IF SUPER^.Step(746, TRUE, 'Step number 746') THEN
    SUPER^.StepCompleteWhen((_runOneStep OR _runAllSteps) AND _finishStep);

    IF _runOneStep THEN
        _runOneStep := FALSE;
        RETURN;
    END_IF
END_IF

IF SUPER^.Step(747, TRUE, 'Step number 747') THEN
    SUPER^.StepCompleteWhen((_runOneStep OR _runAllSteps) AND _finishStep);

    IF _runOneStep THEN
        _runOneStep := FALSE;
        RETURN;
    END_IF
END_IF

IF SUPER^.Step(748, TRUE, 'Step number 748') THEN
    SUPER^.StepCompleteWhen((_runOneStep OR _runAllSteps) AND _finishStep);

    IF _runOneStep THEN
        _runOneStep := FALSE;
        RETURN;
    END_IF
END_IF

IF SUPER^.Step(749, TRUE, 'Step number 749') THEN
    SUPER^.StepCompleteWhen((_runOneStep OR _runAllSteps) AND _finishStep);

    IF _runOneStep THEN
        _runOneStep := FALSE;
        RETURN;
    END_IF
END_IF

IF SUPER^.Step(750, TRUE, 'Step number 750') THEN
    SUPER^.StepCompleteWhen((_runOneStep OR _runAllSteps) AND _finishStep);

    IF _runOneStep THEN
        _runOneStep := FALSE;
        RETURN;
    END_IF
END_IF

IF SUPER^.Step(751, TRUE, 'Step number 751') THEN
    SUPER^.StepCompleteWhen((_runOneStep OR _runAllSteps) AND _finishStep);

    IF _runOneStep THEN
        _runOneStep := FALSE;
        RETURN;
    END_IF
END_IF

IF SUPER^.Step(752, TRUE, 'Step number 752') THEN
    SUPER^.StepCompleteWhen((_runOneStep OR _runAllSteps) AND _finishStep);

    IF _runOneStep THEN
        _runOneStep := FALSE;
        RETURN;
    END_IF
END_IF

IF SUPER^.Step(753, TRUE, 'Step number 753') THEN
    SUPER^.StepCompleteWhen((_runOneStep OR _runAllSteps) AND _finishStep);

    IF _runOneStep THEN
        _runOneStep := FALSE;
        RETURN;
    END_IF
END_IF

IF SUPER^.Step(754, TRUE, 'Step number 754') THEN
    SUPER^.StepCompleteWhen((_runOneStep OR _runAllSteps) AND _finishStep);

    IF _runOneStep THEN
        _runOneStep := FALSE;
        RETURN;
    END_IF
END_IF

IF SUPER^.Step(755, TRUE, 'Step number 755') THEN
    SUPER^.StepCompleteWhen((_runOneStep OR _runAllSteps) AND _finishStep);

    IF _runOneStep THEN
        _runOneStep := FALSE;
        RETURN;
    END_IF
END_IF

IF SUPER^.Step(756, TRUE, 'Step number 756') THEN
    SUPER^.StepCompleteWhen((_runOneStep OR _runAllSteps) AND _finishStep);

    IF _runOneStep THEN
        _runOneStep := FALSE;
        RETURN;
    END_IF
END_IF

IF SUPER^.Step(757, TRUE, 'Step number 757') THEN
    SUPER^.StepCompleteWhen((_runOneStep OR _runAllSteps) AND _finishStep);

    IF _runOneStep THEN
        _runOneStep := FALSE;
        RETURN;
    END_IF
END_IF

IF SUPER^.Step(758, TRUE, 'Step number 758') THEN
    SUPER^.StepCompleteWhen((_runOneStep OR _runAllSteps) AND _finishStep);

    IF _runOneStep THEN
        _runOneStep := FALSE;
        RETURN;
    END_IF
END_IF

IF SUPER^.Step(759, TRUE, 'Step number 759') THEN
    SUPER^.StepCompleteWhen((_runOneStep OR _runAllSteps) AND _finishStep);

    IF _runOneStep THEN
        _runOneStep := FALSE;
        RETURN;
    END_IF
END_IF

IF SUPER^.Step(760, TRUE, 'Step number 760') THEN
    SUPER^.StepCompleteWhen((_runOneStep OR _runAllSteps) AND _finishStep);

    IF _runOneStep THEN
        _runOneStep := FALSE;
        RETURN;
    END_IF
END_IF

IF SUPER^.Step(761, TRUE, 'Step number 761') THEN
    SUPER^.StepCompleteWhen((_runOneStep OR _runAllSteps) AND _finishStep);

    IF _runOneStep THEN
        _runOneStep := FALSE;
        RETURN;
    END_IF
END_IF

IF SUPER^.Step(762, TRUE, 'Step number 762') THEN
    SUPER^.StepCompleteWhen((_runOneStep OR _runAllSteps) AND _finishStep);

    IF _runOneStep THEN
        _runOneStep := FALSE;
        RETURN;
    END_IF
END_IF

IF SUPER^.Step(763, TRUE, 'Step number 763') THEN
    SUPER^.StepCompleteWhen((_runOneStep OR _runAllSteps) AND _finishStep);

    IF _runOneStep THEN
        _runOneStep := FALSE;
        RETURN;
    END_IF
END_IF

IF SUPER^.Step(764, TRUE, 'Step number 764') THEN
    SUPER^.StepCompleteWhen((_runOneStep OR _runAllSteps) AND _finishStep);

    IF _runOneStep THEN
        _runOneStep := FALSE;
        RETURN;
    END_IF
END_IF

IF SUPER^.Step(765, TRUE, 'Step number 765') THEN
    SUPER^.StepCompleteWhen((_runOneStep OR _runAllSteps) AND _finishStep);

    IF _runOneStep THEN
        _runOneStep := FALSE;
        RETURN;
    END_IF
END_IF

IF SUPER^.Step(766, TRUE, 'Step number 766') THEN
    SUPER^.StepCompleteWhen((_runOneStep OR _runAllSteps) AND _finishStep);

    IF _runOneStep THEN
        _runOneStep := FALSE;
        RETURN;
    END_IF
END_IF

IF SUPER^.Step(767, TRUE, 'Step number 767') THEN
    SUPER^.StepCompleteWhen((_runOneStep OR _runAllSteps) AND _finishStep);

    IF _runOneStep THEN
        _runOneStep := FALSE;
        RETURN;
    END_IF
END_IF

IF SUPER^.Step(768, TRUE, 'Step number 768') THEN
    SUPER^.StepCompleteWhen((_runOneStep OR _runAllSteps) AND _finishStep);

    IF _runOneStep THEN
        _runOneStep := FALSE;
        RETURN;
    END_IF
END_IF

IF SUPER^.Step(769, TRUE, 'Step number 769') THEN
    SUPER^.StepCompleteWhen((_runOneStep OR _runAllSteps) AND _finishStep);

    IF _runOneStep THEN
        _runOneStep := FALSE;
        RETURN;
    END_IF
END_IF

IF SUPER^.Step(770, TRUE, 'Step number 770') THEN
    SUPER^.StepCompleteWhen((_runOneStep OR _runAllSteps) AND _finishStep);

    IF _runOneStep THEN
        _runOneStep := FALSE;
        RETURN;
    END_IF
END_IF

IF SUPER^.Step(771, TRUE, 'Step number 771') THEN
    SUPER^.StepCompleteWhen((_runOneStep OR _runAllSteps) AND _finishStep);

    IF _runOneStep THEN
        _runOneStep := FALSE;
        RETURN;
    END_IF
END_IF

IF SUPER^.Step(772, TRUE, 'Step number 772') THEN
    SUPER^.StepCompleteWhen((_runOneStep OR _runAllSteps) AND _finishStep);

    IF _runOneStep THEN
        _runOneStep := FALSE;
        RETURN;
    END_IF
END_IF

IF SUPER^.Step(773, TRUE, 'Step number 773') THEN
    SUPER^.StepCompleteWhen((_runOneStep OR _runAllSteps) AND _finishStep);

    IF _runOneStep THEN
        _runOneStep := FALSE;
        RETURN;
    END_IF
END_IF

IF SUPER^.Step(774, TRUE, 'Step number 774') THEN
    SUPER^.StepCompleteWhen((_runOneStep OR _runAllSteps) AND _finishStep);

    IF _runOneStep THEN
        _runOneStep := FALSE;
        RETURN;
    END_IF
END_IF

IF SUPER^.Step(775, TRUE, 'Step number 775') THEN
    SUPER^.StepCompleteWhen((_runOneStep OR _runAllSteps) AND _finishStep);

    IF _runOneStep THEN
        _runOneStep := FALSE;
        RETURN;
    END_IF
END_IF

IF SUPER^.Step(776, TRUE, 'Step number 776') THEN
    SUPER^.StepCompleteWhen((_runOneStep OR _runAllSteps) AND _finishStep);

    IF _runOneStep THEN
        _runOneStep := FALSE;
        RETURN;
    END_IF
END_IF

IF SUPER^.Step(777, TRUE, 'Step number 777') THEN
    SUPER^.StepCompleteWhen((_runOneStep OR _runAllSteps) AND _finishStep);

    IF _runOneStep THEN
        _runOneStep := FALSE;
        RETURN;
    END_IF
END_IF

IF SUPER^.Step(778, TRUE, 'Step number 778') THEN
    SUPER^.StepCompleteWhen((_runOneStep OR _runAllSteps) AND _finishStep);

    IF _runOneStep THEN
        _runOneStep := FALSE;
        RETURN;
    END_IF
END_IF

IF SUPER^.Step(779, TRUE, 'Step number 779') THEN
    SUPER^.StepCompleteWhen((_runOneStep OR _runAllSteps) AND _finishStep);

    IF _runOneStep THEN
        _runOneStep := FALSE;
        RETURN;
    END_IF
END_IF

IF SUPER^.Step(780, TRUE, 'Step number 780') THEN
    SUPER^.StepCompleteWhen((_runOneStep OR _runAllSteps) AND _finishStep);

    IF _runOneStep THEN
        _runOneStep := FALSE;
        RETURN;
    END_IF
END_IF

IF SUPER^.Step(781, TRUE, 'Step number 781') THEN
    SUPER^.StepCompleteWhen((_runOneStep OR _runAllSteps) AND _finishStep);

    IF _runOneStep THEN
        _runOneStep := FALSE;
        RETURN;
    END_IF
END_IF

IF SUPER^.Step(782, TRUE, 'Step number 782') THEN
    SUPER^.StepCompleteWhen((_runOneStep OR _runAllSteps) AND _finishStep);

    IF _runOneStep THEN
        _runOneStep := FALSE;
        RETURN;
    END_IF
END_IF

IF SUPER^.Step(783, TRUE, 'Step number 783') THEN
    SUPER^.StepCompleteWhen((_runOneStep OR _runAllSteps) AND _finishStep);

    IF _runOneStep THEN
        _runOneStep := FALSE;
        RETURN;
    END_IF
END_IF

IF SUPER^.Step(784, TRUE, 'Step number 784') THEN
    SUPER^.StepCompleteWhen((_runOneStep OR _runAllSteps) AND _finishStep);

    IF _runOneStep THEN
        _runOneStep := FALSE;
        RETURN;
    END_IF
END_IF

IF SUPER^.Step(785, TRUE, 'Step number 785') THEN
    SUPER^.StepCompleteWhen((_runOneStep OR _runAllSteps) AND _finishStep);

    IF _runOneStep THEN
        _runOneStep := FALSE;
        RETURN;
    END_IF
END_IF

IF SUPER^.Step(786, TRUE, 'Step number 786') THEN
    SUPER^.StepCompleteWhen((_runOneStep OR _runAllSteps) AND _finishStep);

    IF _runOneStep THEN
        _runOneStep := FALSE;
        RETURN;
    END_IF
END_IF

IF SUPER^.Step(787, TRUE, 'Step number 787') THEN
    SUPER^.StepCompleteWhen((_runOneStep OR _runAllSteps) AND _finishStep);

    IF _runOneStep THEN
        _runOneStep := FALSE;
        RETURN;
    END_IF
END_IF

IF SUPER^.Step(788, TRUE, 'Step number 788') THEN
    SUPER^.StepCompleteWhen((_runOneStep OR _runAllSteps) AND _finishStep);

    IF _runOneStep THEN
        _runOneStep := FALSE;
        RETURN;
    END_IF
END_IF

IF SUPER^.Step(789, TRUE, 'Step number 789') THEN
    SUPER^.StepCompleteWhen((_runOneStep OR _runAllSteps) AND _finishStep);

    IF _runOneStep THEN
        _runOneStep := FALSE;
        RETURN;
    END_IF
END_IF

IF SUPER^.Step(790, TRUE, 'Step number 790') THEN
    SUPER^.StepCompleteWhen((_runOneStep OR _runAllSteps) AND _finishStep);

    IF _runOneStep THEN
        _runOneStep := FALSE;
        RETURN;
    END_IF
END_IF

IF SUPER^.Step(791, TRUE, 'Step number 791') THEN
    SUPER^.StepCompleteWhen((_runOneStep OR _runAllSteps) AND _finishStep);

    IF _runOneStep THEN
        _runOneStep := FALSE;
        RETURN;
    END_IF
END_IF

IF SUPER^.Step(792, TRUE, 'Step number 792') THEN
    SUPER^.StepCompleteWhen((_runOneStep OR _runAllSteps) AND _finishStep);

    IF _runOneStep THEN
        _runOneStep := FALSE;
        RETURN;
    END_IF
END_IF

IF SUPER^.Step(793, TRUE, 'Step number 793') THEN
    SUPER^.StepCompleteWhen((_runOneStep OR _runAllSteps) AND _finishStep);

    IF _runOneStep THEN
        _runOneStep := FALSE;
        RETURN;
    END_IF
END_IF

IF SUPER^.Step(794, TRUE, 'Step number 794') THEN
    SUPER^.StepCompleteWhen((_runOneStep OR _runAllSteps) AND _finishStep);

    IF _runOneStep THEN
        _runOneStep := FALSE;
        RETURN;
    END_IF
END_IF

IF SUPER^.Step(795, TRUE, 'Step number 795') THEN
    SUPER^.StepCompleteWhen((_runOneStep OR _runAllSteps) AND _finishStep);

    IF _runOneStep THEN
        _runOneStep := FALSE;
        RETURN;
    END_IF
END_IF

IF SUPER^.Step(796, TRUE, 'Step number 796') THEN
    SUPER^.StepCompleteWhen((_runOneStep OR _runAllSteps) AND _finishStep);

    IF _runOneStep THEN
        _runOneStep := FALSE;
        RETURN;
    END_IF
END_IF

IF SUPER^.Step(797, TRUE, 'Step number 797') THEN
    SUPER^.StepCompleteWhen((_runOneStep OR _runAllSteps) AND _finishStep);

    IF _runOneStep THEN
        _runOneStep := FALSE;
        RETURN;
    END_IF
END_IF

IF SUPER^.Step(798, TRUE, 'Step number 798') THEN
    SUPER^.StepCompleteWhen((_runOneStep OR _runAllSteps) AND _finishStep);

    IF _runOneStep THEN
        _runOneStep := FALSE;
        RETURN;
    END_IF
END_IF

IF SUPER^.Step(799, TRUE, 'Step number 799') THEN
    SUPER^.StepCompleteWhen((_runOneStep OR _runAllSteps) AND _finishStep);

    IF _runOneStep THEN
        _runOneStep := FALSE;
        RETURN;
    END_IF
END_IF

IF SUPER^.Step(800, TRUE, 'Step number 800') THEN
    SUPER^.StepCompleteWhen((_runOneStep OR _runAllSteps) AND _finishStep);

    IF _runOneStep THEN
        _runOneStep := FALSE;
        RETURN;
    END_IF
END_IF

IF SUPER^.Step(801, TRUE, 'Step number 801') THEN
    SUPER^.StepCompleteWhen((_runOneStep OR _runAllSteps) AND _finishStep);

    IF _runOneStep THEN
        _runOneStep := FALSE;
        RETURN;
    END_IF
END_IF

IF SUPER^.Step(802, TRUE, 'Step number 802') THEN
    SUPER^.StepCompleteWhen((_runOneStep OR _runAllSteps) AND _finishStep);

    IF _runOneStep THEN
        _runOneStep := FALSE;
        RETURN;
    END_IF
END_IF

IF SUPER^.Step(803, TRUE, 'Step number 803') THEN
    SUPER^.StepCompleteWhen((_runOneStep OR _runAllSteps) AND _finishStep);

    IF _runOneStep THEN
        _runOneStep := FALSE;
        RETURN;
    END_IF
END_IF

IF SUPER^.Step(804, TRUE, 'Step number 804') THEN
    SUPER^.StepCompleteWhen((_runOneStep OR _runAllSteps) AND _finishStep);

    IF _runOneStep THEN
        _runOneStep := FALSE;
        RETURN;
    END_IF
END_IF

IF SUPER^.Step(805, TRUE, 'Step number 805') THEN
    SUPER^.StepCompleteWhen((_runOneStep OR _runAllSteps) AND _finishStep);

    IF _runOneStep THEN
        _runOneStep := FALSE;
        RETURN;
    END_IF
END_IF

IF SUPER^.Step(806, TRUE, 'Step number 806') THEN
    SUPER^.StepCompleteWhen((_runOneStep OR _runAllSteps) AND _finishStep);

    IF _runOneStep THEN
        _runOneStep := FALSE;
        RETURN;
    END_IF
END_IF

IF SUPER^.Step(807, TRUE, 'Step number 807') THEN
    SUPER^.StepCompleteWhen((_runOneStep OR _runAllSteps) AND _finishStep);

    IF _runOneStep THEN
        _runOneStep := FALSE;
        RETURN;
    END_IF
END_IF

IF SUPER^.Step(808, TRUE, 'Step number 808') THEN
    SUPER^.StepCompleteWhen((_runOneStep OR _runAllSteps) AND _finishStep);

    IF _runOneStep THEN
        _runOneStep := FALSE;
        RETURN;
    END_IF
END_IF

IF SUPER^.Step(809, TRUE, 'Step number 809') THEN
    SUPER^.StepCompleteWhen((_runOneStep OR _runAllSteps) AND _finishStep);

    IF _runOneStep THEN
        _runOneStep := FALSE;
        RETURN;
    END_IF
END_IF

IF SUPER^.Step(810, TRUE, 'Step number 810') THEN
    SUPER^.StepCompleteWhen((_runOneStep OR _runAllSteps) AND _finishStep);

    IF _runOneStep THEN
        _runOneStep := FALSE;
        RETURN;
    END_IF
END_IF

IF SUPER^.Step(811, TRUE, 'Step number 811') THEN
    SUPER^.StepCompleteWhen((_runOneStep OR _runAllSteps) AND _finishStep);

    IF _runOneStep THEN
        _runOneStep := FALSE;
        RETURN;
    END_IF
END_IF

IF SUPER^.Step(812, TRUE, 'Step number 812') THEN
    SUPER^.StepCompleteWhen((_runOneStep OR _runAllSteps) AND _finishStep);

    IF _runOneStep THEN
        _runOneStep := FALSE;
        RETURN;
    END_IF
END_IF

IF SUPER^.Step(813, TRUE, 'Step number 813') THEN
    SUPER^.StepCompleteWhen((_runOneStep OR _runAllSteps) AND _finishStep);

    IF _runOneStep THEN
        _runOneStep := FALSE;
        RETURN;
    END_IF
END_IF

IF SUPER^.Step(814, TRUE, 'Step number 814') THEN
    SUPER^.StepCompleteWhen((_runOneStep OR _runAllSteps) AND _finishStep);

    IF _runOneStep THEN
        _runOneStep := FALSE;
        RETURN;
    END_IF
END_IF

IF SUPER^.Step(815, TRUE, 'Step number 815') THEN
    SUPER^.StepCompleteWhen((_runOneStep OR _runAllSteps) AND _finishStep);

    IF _runOneStep THEN
        _runOneStep := FALSE;
        RETURN;
    END_IF
END_IF

IF SUPER^.Step(816, TRUE, 'Step number 816') THEN
    SUPER^.StepCompleteWhen((_runOneStep OR _runAllSteps) AND _finishStep);

    IF _runOneStep THEN
        _runOneStep := FALSE;
        RETURN;
    END_IF
END_IF

IF SUPER^.Step(817, TRUE, 'Step number 817') THEN
    SUPER^.StepCompleteWhen((_runOneStep OR _runAllSteps) AND _finishStep);

    IF _runOneStep THEN
        _runOneStep := FALSE;
        RETURN;
    END_IF
END_IF

IF SUPER^.Step(818, TRUE, 'Step number 818') THEN
    SUPER^.StepCompleteWhen((_runOneStep OR _runAllSteps) AND _finishStep);

    IF _runOneStep THEN
        _runOneStep := FALSE;
        RETURN;
    END_IF
END_IF

IF SUPER^.Step(819, TRUE, 'Step number 819') THEN
    SUPER^.StepCompleteWhen((_runOneStep OR _runAllSteps) AND _finishStep);

    IF _runOneStep THEN
        _runOneStep := FALSE;
        RETURN;
    END_IF
END_IF

IF SUPER^.Step(820, TRUE, 'Step number 820') THEN
    SUPER^.StepCompleteWhen((_runOneStep OR _runAllSteps) AND _finishStep);

    IF _runOneStep THEN
        _runOneStep := FALSE;
        RETURN;
    END_IF
END_IF

IF SUPER^.Step(821, TRUE, 'Step number 821') THEN
    SUPER^.StepCompleteWhen((_runOneStep OR _runAllSteps) AND _finishStep);

    IF _runOneStep THEN
        _runOneStep := FALSE;
        RETURN;
    END_IF
END_IF

IF SUPER^.Step(822, TRUE, 'Step number 822') THEN
    SUPER^.StepCompleteWhen((_runOneStep OR _runAllSteps) AND _finishStep);

    IF _runOneStep THEN
        _runOneStep := FALSE;
        RETURN;
    END_IF
END_IF

IF SUPER^.Step(823, TRUE, 'Step number 823') THEN
    SUPER^.StepCompleteWhen((_runOneStep OR _runAllSteps) AND _finishStep);

    IF _runOneStep THEN
        _runOneStep := FALSE;
        RETURN;
    END_IF
END_IF

IF SUPER^.Step(824, TRUE, 'Step number 824') THEN
    SUPER^.StepCompleteWhen((_runOneStep OR _runAllSteps) AND _finishStep);

    IF _runOneStep THEN
        _runOneStep := FALSE;
        RETURN;
    END_IF
END_IF

IF SUPER^.Step(825, TRUE, 'Step number 825') THEN
    SUPER^.StepCompleteWhen((_runOneStep OR _runAllSteps) AND _finishStep);

    IF _runOneStep THEN
        _runOneStep := FALSE;
        RETURN;
    END_IF
END_IF

IF SUPER^.Step(826, TRUE, 'Step number 826') THEN
    SUPER^.StepCompleteWhen((_runOneStep OR _runAllSteps) AND _finishStep);

    IF _runOneStep THEN
        _runOneStep := FALSE;
        RETURN;
    END_IF
END_IF

IF SUPER^.Step(827, TRUE, 'Step number 827') THEN
    SUPER^.StepCompleteWhen((_runOneStep OR _runAllSteps) AND _finishStep);

    IF _runOneStep THEN
        _runOneStep := FALSE;
        RETURN;
    END_IF
END_IF

IF SUPER^.Step(828, TRUE, 'Step number 828') THEN
    SUPER^.StepCompleteWhen((_runOneStep OR _runAllSteps) AND _finishStep);

    IF _runOneStep THEN
        _runOneStep := FALSE;
        RETURN;
    END_IF
END_IF

IF SUPER^.Step(829, TRUE, 'Step number 829') THEN
    SUPER^.StepCompleteWhen((_runOneStep OR _runAllSteps) AND _finishStep);

    IF _runOneStep THEN
        _runOneStep := FALSE;
        RETURN;
    END_IF
END_IF

IF SUPER^.Step(830, TRUE, 'Step number 830') THEN
    SUPER^.StepCompleteWhen((_runOneStep OR _runAllSteps) AND _finishStep);

    IF _runOneStep THEN
        _runOneStep := FALSE;
        RETURN;
    END_IF
END_IF

IF SUPER^.Step(831, TRUE, 'Step number 831') THEN
    SUPER^.StepCompleteWhen((_runOneStep OR _runAllSteps) AND _finishStep);

    IF _runOneStep THEN
        _runOneStep := FALSE;
        RETURN;
    END_IF
END_IF

IF SUPER^.Step(832, TRUE, 'Step number 832') THEN
    SUPER^.StepCompleteWhen((_runOneStep OR _runAllSteps) AND _finishStep);

    IF _runOneStep THEN
        _runOneStep := FALSE;
        RETURN;
    END_IF
END_IF

IF SUPER^.Step(833, TRUE, 'Step number 833') THEN
    SUPER^.StepCompleteWhen((_runOneStep OR _runAllSteps) AND _finishStep);

    IF _runOneStep THEN
        _runOneStep := FALSE;
        RETURN;
    END_IF
END_IF

IF SUPER^.Step(834, TRUE, 'Step number 834') THEN
    SUPER^.StepCompleteWhen((_runOneStep OR _runAllSteps) AND _finishStep);

    IF _runOneStep THEN
        _runOneStep := FALSE;
        RETURN;
    END_IF
END_IF

IF SUPER^.Step(835, TRUE, 'Step number 835') THEN
    SUPER^.StepCompleteWhen((_runOneStep OR _runAllSteps) AND _finishStep);

    IF _runOneStep THEN
        _runOneStep := FALSE;
        RETURN;
    END_IF
END_IF

IF SUPER^.Step(836, TRUE, 'Step number 836') THEN
    SUPER^.StepCompleteWhen((_runOneStep OR _runAllSteps) AND _finishStep);

    IF _runOneStep THEN
        _runOneStep := FALSE;
        RETURN;
    END_IF
END_IF

IF SUPER^.Step(837, TRUE, 'Step number 837') THEN
    SUPER^.StepCompleteWhen((_runOneStep OR _runAllSteps) AND _finishStep);

    IF _runOneStep THEN
        _runOneStep := FALSE;
        RETURN;
    END_IF
END_IF

IF SUPER^.Step(838, TRUE, 'Step number 838') THEN
    SUPER^.StepCompleteWhen((_runOneStep OR _runAllSteps) AND _finishStep);

    IF _runOneStep THEN
        _runOneStep := FALSE;
        RETURN;
    END_IF
END_IF

IF SUPER^.Step(839, TRUE, 'Step number 839') THEN
    SUPER^.StepCompleteWhen((_runOneStep OR _runAllSteps) AND _finishStep);

    IF _runOneStep THEN
        _runOneStep := FALSE;
        RETURN;
    END_IF
END_IF

IF SUPER^.Step(840, TRUE, 'Step number 840') THEN
    SUPER^.StepCompleteWhen((_runOneStep OR _runAllSteps) AND _finishStep);

    IF _runOneStep THEN
        _runOneStep := FALSE;
        RETURN;
    END_IF
END_IF

IF SUPER^.Step(841, TRUE, 'Step number 841') THEN
    SUPER^.StepCompleteWhen((_runOneStep OR _runAllSteps) AND _finishStep);

    IF _runOneStep THEN
        _runOneStep := FALSE;
        RETURN;
    END_IF
END_IF

IF SUPER^.Step(842, TRUE, 'Step number 842') THEN
    SUPER^.StepCompleteWhen((_runOneStep OR _runAllSteps) AND _finishStep);

    IF _runOneStep THEN
        _runOneStep := FALSE;
        RETURN;
    END_IF
END_IF

IF SUPER^.Step(843, TRUE, 'Step number 843') THEN
    SUPER^.StepCompleteWhen((_runOneStep OR _runAllSteps) AND _finishStep);

    IF _runOneStep THEN
        _runOneStep := FALSE;
        RETURN;
    END_IF
END_IF

IF SUPER^.Step(844, TRUE, 'Step number 844') THEN
    SUPER^.StepCompleteWhen((_runOneStep OR _runAllSteps) AND _finishStep);

    IF _runOneStep THEN
        _runOneStep := FALSE;
        RETURN;
    END_IF
END_IF

IF SUPER^.Step(845, TRUE, 'Step number 845') THEN
    SUPER^.StepCompleteWhen((_runOneStep OR _runAllSteps) AND _finishStep);

    IF _runOneStep THEN
        _runOneStep := FALSE;
        RETURN;
    END_IF
END_IF

IF SUPER^.Step(846, TRUE, 'Step number 846') THEN
    SUPER^.StepCompleteWhen((_runOneStep OR _runAllSteps) AND _finishStep);

    IF _runOneStep THEN
        _runOneStep := FALSE;
        RETURN;
    END_IF
END_IF

IF SUPER^.Step(847, TRUE, 'Step number 847') THEN
    SUPER^.StepCompleteWhen((_runOneStep OR _runAllSteps) AND _finishStep);

    IF _runOneStep THEN
        _runOneStep := FALSE;
        RETURN;
    END_IF
END_IF

IF SUPER^.Step(848, TRUE, 'Step number 848') THEN
    SUPER^.StepCompleteWhen((_runOneStep OR _runAllSteps) AND _finishStep);

    IF _runOneStep THEN
        _runOneStep := FALSE;
        RETURN;
    END_IF
END_IF

IF SUPER^.Step(849, TRUE, 'Step number 849') THEN
    SUPER^.StepCompleteWhen((_runOneStep OR _runAllSteps) AND _finishStep);

    IF _runOneStep THEN
        _runOneStep := FALSE;
        RETURN;
    END_IF
END_IF

IF SUPER^.Step(850, TRUE, 'Step number 850') THEN
    SUPER^.StepCompleteWhen((_runOneStep OR _runAllSteps) AND _finishStep);

    IF _runOneStep THEN
        _runOneStep := FALSE;
        RETURN;
    END_IF
END_IF

IF SUPER^.Step(851, TRUE, 'Step number 851') THEN
    SUPER^.StepCompleteWhen((_runOneStep OR _runAllSteps) AND _finishStep);

    IF _runOneStep THEN
        _runOneStep := FALSE;
        RETURN;
    END_IF
END_IF

IF SUPER^.Step(852, TRUE, 'Step number 852') THEN
    SUPER^.StepCompleteWhen((_runOneStep OR _runAllSteps) AND _finishStep);

    IF _runOneStep THEN
        _runOneStep := FALSE;
        RETURN;
    END_IF
END_IF

IF SUPER^.Step(853, TRUE, 'Step number 853') THEN
    SUPER^.StepCompleteWhen((_runOneStep OR _runAllSteps) AND _finishStep);

    IF _runOneStep THEN
        _runOneStep := FALSE;
        RETURN;
    END_IF
END_IF

IF SUPER^.Step(854, TRUE, 'Step number 854') THEN
    SUPER^.StepCompleteWhen((_runOneStep OR _runAllSteps) AND _finishStep);

    IF _runOneStep THEN
        _runOneStep := FALSE;
        RETURN;
    END_IF
END_IF

IF SUPER^.Step(855, TRUE, 'Step number 855') THEN
    SUPER^.StepCompleteWhen((_runOneStep OR _runAllSteps) AND _finishStep);

    IF _runOneStep THEN
        _runOneStep := FALSE;
        RETURN;
    END_IF
END_IF

IF SUPER^.Step(856, TRUE, 'Step number 856') THEN
    SUPER^.StepCompleteWhen((_runOneStep OR _runAllSteps) AND _finishStep);

    IF _runOneStep THEN
        _runOneStep := FALSE;
        RETURN;
    END_IF
END_IF

IF SUPER^.Step(857, TRUE, 'Step number 857') THEN
    SUPER^.StepCompleteWhen((_runOneStep OR _runAllSteps) AND _finishStep);

    IF _runOneStep THEN
        _runOneStep := FALSE;
        RETURN;
    END_IF
END_IF

IF SUPER^.Step(858, TRUE, 'Step number 858') THEN
    SUPER^.StepCompleteWhen((_runOneStep OR _runAllSteps) AND _finishStep);

    IF _runOneStep THEN
        _runOneStep := FALSE;
        RETURN;
    END_IF
END_IF

IF SUPER^.Step(859, TRUE, 'Step number 859') THEN
    SUPER^.StepCompleteWhen((_runOneStep OR _runAllSteps) AND _finishStep);

    IF _runOneStep THEN
        _runOneStep := FALSE;
        RETURN;
    END_IF
END_IF

IF SUPER^.Step(860, TRUE, 'Step number 860') THEN
    SUPER^.StepCompleteWhen((_runOneStep OR _runAllSteps) AND _finishStep);

    IF _runOneStep THEN
        _runOneStep := FALSE;
        RETURN;
    END_IF
END_IF

IF SUPER^.Step(861, TRUE, 'Step number 861') THEN
    SUPER^.StepCompleteWhen((_runOneStep OR _runAllSteps) AND _finishStep);

    IF _runOneStep THEN
        _runOneStep := FALSE;
        RETURN;
    END_IF
END_IF

IF SUPER^.Step(862, TRUE, 'Step number 862') THEN
    SUPER^.StepCompleteWhen((_runOneStep OR _runAllSteps) AND _finishStep);

    IF _runOneStep THEN
        _runOneStep := FALSE;
        RETURN;
    END_IF
END_IF

IF SUPER^.Step(863, TRUE, 'Step number 863') THEN
    SUPER^.StepCompleteWhen((_runOneStep OR _runAllSteps) AND _finishStep);

    IF _runOneStep THEN
        _runOneStep := FALSE;
        RETURN;
    END_IF
END_IF

IF SUPER^.Step(864, TRUE, 'Step number 864') THEN
    SUPER^.StepCompleteWhen((_runOneStep OR _runAllSteps) AND _finishStep);

    IF _runOneStep THEN
        _runOneStep := FALSE;
        RETURN;
    END_IF
END_IF

IF SUPER^.Step(865, TRUE, 'Step number 865') THEN
    SUPER^.StepCompleteWhen((_runOneStep OR _runAllSteps) AND _finishStep);

    IF _runOneStep THEN
        _runOneStep := FALSE;
        RETURN;
    END_IF
END_IF

IF SUPER^.Step(866, TRUE, 'Step number 866') THEN
    SUPER^.StepCompleteWhen((_runOneStep OR _runAllSteps) AND _finishStep);

    IF _runOneStep THEN
        _runOneStep := FALSE;
        RETURN;
    END_IF
END_IF

IF SUPER^.Step(867, TRUE, 'Step number 867') THEN
    SUPER^.StepCompleteWhen((_runOneStep OR _runAllSteps) AND _finishStep);

    IF _runOneStep THEN
        _runOneStep := FALSE;
        RETURN;
    END_IF
END_IF

IF SUPER^.Step(868, TRUE, 'Step number 868') THEN
    SUPER^.StepCompleteWhen((_runOneStep OR _runAllSteps) AND _finishStep);

    IF _runOneStep THEN
        _runOneStep := FALSE;
        RETURN;
    END_IF
END_IF

IF SUPER^.Step(869, TRUE, 'Step number 869') THEN
    SUPER^.StepCompleteWhen((_runOneStep OR _runAllSteps) AND _finishStep);

    IF _runOneStep THEN
        _runOneStep := FALSE;
        RETURN;
    END_IF
END_IF

IF SUPER^.Step(870, TRUE, 'Step number 870') THEN
    SUPER^.StepCompleteWhen((_runOneStep OR _runAllSteps) AND _finishStep);

    IF _runOneStep THEN
        _runOneStep := FALSE;
        RETURN;
    END_IF
END_IF

IF SUPER^.Step(871, TRUE, 'Step number 871') THEN
    SUPER^.StepCompleteWhen((_runOneStep OR _runAllSteps) AND _finishStep);

    IF _runOneStep THEN
        _runOneStep := FALSE;
        RETURN;
    END_IF
END_IF

IF SUPER^.Step(872, TRUE, 'Step number 872') THEN
    SUPER^.StepCompleteWhen((_runOneStep OR _runAllSteps) AND _finishStep);

    IF _runOneStep THEN
        _runOneStep := FALSE;
        RETURN;
    END_IF
END_IF

IF SUPER^.Step(873, TRUE, 'Step number 873') THEN
    SUPER^.StepCompleteWhen((_runOneStep OR _runAllSteps) AND _finishStep);

    IF _runOneStep THEN
        _runOneStep := FALSE;
        RETURN;
    END_IF
END_IF

IF SUPER^.Step(874, TRUE, 'Step number 874') THEN
    SUPER^.StepCompleteWhen((_runOneStep OR _runAllSteps) AND _finishStep);

    IF _runOneStep THEN
        _runOneStep := FALSE;
        RETURN;
    END_IF
END_IF

IF SUPER^.Step(875, TRUE, 'Step number 875') THEN
    SUPER^.StepCompleteWhen((_runOneStep OR _runAllSteps) AND _finishStep);

    IF _runOneStep THEN
        _runOneStep := FALSE;
        RETURN;
    END_IF
END_IF

IF SUPER^.Step(876, TRUE, 'Step number 876') THEN
    SUPER^.StepCompleteWhen((_runOneStep OR _runAllSteps) AND _finishStep);

    IF _runOneStep THEN
        _runOneStep := FALSE;
        RETURN;
    END_IF
END_IF

IF SUPER^.Step(877, TRUE, 'Step number 877') THEN
    SUPER^.StepCompleteWhen((_runOneStep OR _runAllSteps) AND _finishStep);

    IF _runOneStep THEN
        _runOneStep := FALSE;
        RETURN;
    END_IF
END_IF

IF SUPER^.Step(878, TRUE, 'Step number 878') THEN
    SUPER^.StepCompleteWhen((_runOneStep OR _runAllSteps) AND _finishStep);

    IF _runOneStep THEN
        _runOneStep := FALSE;
        RETURN;
    END_IF
END_IF

IF SUPER^.Step(879, TRUE, 'Step number 879') THEN
    SUPER^.StepCompleteWhen((_runOneStep OR _runAllSteps) AND _finishStep);

    IF _runOneStep THEN
        _runOneStep := FALSE;
        RETURN;
    END_IF
END_IF

IF SUPER^.Step(880, TRUE, 'Step number 880') THEN
    SUPER^.StepCompleteWhen((_runOneStep OR _runAllSteps) AND _finishStep);

    IF _runOneStep THEN
        _runOneStep := FALSE;
        RETURN;
    END_IF
END_IF

IF SUPER^.Step(881, TRUE, 'Step number 881') THEN
    SUPER^.StepCompleteWhen((_runOneStep OR _runAllSteps) AND _finishStep);

    IF _runOneStep THEN
        _runOneStep := FALSE;
        RETURN;
    END_IF
END_IF

IF SUPER^.Step(882, TRUE, 'Step number 882') THEN
    SUPER^.StepCompleteWhen((_runOneStep OR _runAllSteps) AND _finishStep);

    IF _runOneStep THEN
        _runOneStep := FALSE;
        RETURN;
    END_IF
END_IF

IF SUPER^.Step(883, TRUE, 'Step number 883') THEN
    SUPER^.StepCompleteWhen((_runOneStep OR _runAllSteps) AND _finishStep);

    IF _runOneStep THEN
        _runOneStep := FALSE;
        RETURN;
    END_IF
END_IF

IF SUPER^.Step(884, TRUE, 'Step number 884') THEN
    SUPER^.StepCompleteWhen((_runOneStep OR _runAllSteps) AND _finishStep);

    IF _runOneStep THEN
        _runOneStep := FALSE;
        RETURN;
    END_IF
END_IF

IF SUPER^.Step(885, TRUE, 'Step number 885') THEN
    SUPER^.StepCompleteWhen((_runOneStep OR _runAllSteps) AND _finishStep);

    IF _runOneStep THEN
        _runOneStep := FALSE;
        RETURN;
    END_IF
END_IF

IF SUPER^.Step(886, TRUE, 'Step number 886') THEN
    SUPER^.StepCompleteWhen((_runOneStep OR _runAllSteps) AND _finishStep);

    IF _runOneStep THEN
        _runOneStep := FALSE;
        RETURN;
    END_IF
END_IF

IF SUPER^.Step(887, TRUE, 'Step number 887') THEN
    SUPER^.StepCompleteWhen((_runOneStep OR _runAllSteps) AND _finishStep);

    IF _runOneStep THEN
        _runOneStep := FALSE;
        RETURN;
    END_IF
END_IF

IF SUPER^.Step(888, TRUE, 'Step number 888') THEN
    SUPER^.StepCompleteWhen((_runOneStep OR _runAllSteps) AND _finishStep);

    IF _runOneStep THEN
        _runOneStep := FALSE;
        RETURN;
    END_IF
END_IF

IF SUPER^.Step(889, TRUE, 'Step number 889') THEN
    SUPER^.StepCompleteWhen((_runOneStep OR _runAllSteps) AND _finishStep);

    IF _runOneStep THEN
        _runOneStep := FALSE;
        RETURN;
    END_IF
END_IF

IF SUPER^.Step(890, TRUE, 'Step number 890') THEN
    SUPER^.StepCompleteWhen((_runOneStep OR _runAllSteps) AND _finishStep);

    IF _runOneStep THEN
        _runOneStep := FALSE;
        RETURN;
    END_IF
END_IF

IF SUPER^.Step(891, TRUE, 'Step number 891') THEN
    SUPER^.StepCompleteWhen((_runOneStep OR _runAllSteps) AND _finishStep);

    IF _runOneStep THEN
        _runOneStep := FALSE;
        RETURN;
    END_IF
END_IF

IF SUPER^.Step(892, TRUE, 'Step number 892') THEN
    SUPER^.StepCompleteWhen((_runOneStep OR _runAllSteps) AND _finishStep);

    IF _runOneStep THEN
        _runOneStep := FALSE;
        RETURN;
    END_IF
END_IF

IF SUPER^.Step(893, TRUE, 'Step number 893') THEN
    SUPER^.StepCompleteWhen((_runOneStep OR _runAllSteps) AND _finishStep);

    IF _runOneStep THEN
        _runOneStep := FALSE;
        RETURN;
    END_IF
END_IF

IF SUPER^.Step(894, TRUE, 'Step number 894') THEN
    SUPER^.StepCompleteWhen((_runOneStep OR _runAllSteps) AND _finishStep);

    IF _runOneStep THEN
        _runOneStep := FALSE;
        RETURN;
    END_IF
END_IF

IF SUPER^.Step(895, TRUE, 'Step number 895') THEN
    SUPER^.StepCompleteWhen((_runOneStep OR _runAllSteps) AND _finishStep);

    IF _runOneStep THEN
        _runOneStep := FALSE;
        RETURN;
    END_IF
END_IF

IF SUPER^.Step(896, TRUE, 'Step number 896') THEN
    SUPER^.StepCompleteWhen((_runOneStep OR _runAllSteps) AND _finishStep);

    IF _runOneStep THEN
        _runOneStep := FALSE;
        RETURN;
    END_IF
END_IF

IF SUPER^.Step(897, TRUE, 'Step number 897') THEN
    SUPER^.StepCompleteWhen((_runOneStep OR _runAllSteps) AND _finishStep);

    IF _runOneStep THEN
        _runOneStep := FALSE;
        RETURN;
    END_IF
END_IF

IF SUPER^.Step(898, TRUE, 'Step number 898') THEN
    SUPER^.StepCompleteWhen((_runOneStep OR _runAllSteps) AND _finishStep);

    IF _runOneStep THEN
        _runOneStep := FALSE;
        RETURN;
    END_IF
END_IF

IF SUPER^.Step(899, TRUE, 'Step number 899') THEN
    SUPER^.StepCompleteWhen((_runOneStep OR _runAllSteps) AND _finishStep);

    IF _runOneStep THEN
        _runOneStep := FALSE;
        RETURN;
    END_IF
END_IF

IF SUPER^.Step(900, TRUE, 'Step number 900') THEN
    SUPER^.StepCompleteWhen((_runOneStep OR _runAllSteps) AND _finishStep);

    IF _runOneStep THEN
        _runOneStep := FALSE;
        RETURN;
    END_IF
END_IF

IF SUPER^.Step(901, TRUE, 'Step number 901') THEN
    SUPER^.StepCompleteWhen((_runOneStep OR _runAllSteps) AND _finishStep);

    IF _runOneStep THEN
        _runOneStep := FALSE;
        RETURN;
    END_IF
END_IF

IF SUPER^.Step(902, TRUE, 'Step number 902') THEN
    SUPER^.StepCompleteWhen((_runOneStep OR _runAllSteps) AND _finishStep);

    IF _runOneStep THEN
        _runOneStep := FALSE;
        RETURN;
    END_IF
END_IF

IF SUPER^.Step(903, TRUE, 'Step number 903') THEN
    SUPER^.StepCompleteWhen((_runOneStep OR _runAllSteps) AND _finishStep);

    IF _runOneStep THEN
        _runOneStep := FALSE;
        RETURN;
    END_IF
END_IF

IF SUPER^.Step(904, TRUE, 'Step number 904') THEN
    SUPER^.StepCompleteWhen((_runOneStep OR _runAllSteps) AND _finishStep);

    IF _runOneStep THEN
        _runOneStep := FALSE;
        RETURN;
    END_IF
END_IF

IF SUPER^.Step(905, TRUE, 'Step number 905') THEN
    SUPER^.StepCompleteWhen((_runOneStep OR _runAllSteps) AND _finishStep);

    IF _runOneStep THEN
        _runOneStep := FALSE;
        RETURN;
    END_IF
END_IF

IF SUPER^.Step(906, TRUE, 'Step number 906') THEN
    SUPER^.StepCompleteWhen((_runOneStep OR _runAllSteps) AND _finishStep);

    IF _runOneStep THEN
        _runOneStep := FALSE;
        RETURN;
    END_IF
END_IF

IF SUPER^.Step(907, TRUE, 'Step number 907') THEN
    SUPER^.StepCompleteWhen((_runOneStep OR _runAllSteps) AND _finishStep);

    IF _runOneStep THEN
        _runOneStep := FALSE;
        RETURN;
    END_IF
END_IF

IF SUPER^.Step(908, TRUE, 'Step number 908') THEN
    SUPER^.StepCompleteWhen((_runOneStep OR _runAllSteps) AND _finishStep);

    IF _runOneStep THEN
        _runOneStep := FALSE;
        RETURN;
    END_IF
END_IF

IF SUPER^.Step(909, TRUE, 'Step number 909') THEN
    SUPER^.StepCompleteWhen((_runOneStep OR _runAllSteps) AND _finishStep);

    IF _runOneStep THEN
        _runOneStep := FALSE;
        RETURN;
    END_IF
END_IF

IF SUPER^.Step(910, TRUE, 'Step number 910') THEN
    SUPER^.StepCompleteWhen((_runOneStep OR _runAllSteps) AND _finishStep);

    IF _runOneStep THEN
        _runOneStep := FALSE;
        RETURN;
    END_IF
END_IF

IF SUPER^.Step(911, TRUE, 'Step number 911') THEN
    SUPER^.StepCompleteWhen((_runOneStep OR _runAllSteps) AND _finishStep);

    IF _runOneStep THEN
        _runOneStep := FALSE;
        RETURN;
    END_IF
END_IF

IF SUPER^.Step(912, TRUE, 'Step number 912') THEN
    SUPER^.StepCompleteWhen((_runOneStep OR _runAllSteps) AND _finishStep);

    IF _runOneStep THEN
        _runOneStep := FALSE;
        RETURN;
    END_IF
END_IF

IF SUPER^.Step(913, TRUE, 'Step number 913') THEN
    SUPER^.StepCompleteWhen((_runOneStep OR _runAllSteps) AND _finishStep);

    IF _runOneStep THEN
        _runOneStep := FALSE;
        RETURN;
    END_IF
END_IF

IF SUPER^.Step(914, TRUE, 'Step number 914') THEN
    SUPER^.StepCompleteWhen((_runOneStep OR _runAllSteps) AND _finishStep);

    IF _runOneStep THEN
        _runOneStep := FALSE;
        RETURN;
    END_IF
END_IF

IF SUPER^.Step(915, TRUE, 'Step number 915') THEN
    SUPER^.StepCompleteWhen((_runOneStep OR _runAllSteps) AND _finishStep);

    IF _runOneStep THEN
        _runOneStep := FALSE;
        RETURN;
    END_IF
END_IF

IF SUPER^.Step(916, TRUE, 'Step number 916') THEN
    SUPER^.StepCompleteWhen((_runOneStep OR _runAllSteps) AND _finishStep);

    IF _runOneStep THEN
        _runOneStep := FALSE;
        RETURN;
    END_IF
END_IF

IF SUPER^.Step(917, TRUE, 'Step number 917') THEN
    SUPER^.StepCompleteWhen((_runOneStep OR _runAllSteps) AND _finishStep);

    IF _runOneStep THEN
        _runOneStep := FALSE;
        RETURN;
    END_IF
END_IF

IF SUPER^.Step(918, TRUE, 'Step number 918') THEN
    SUPER^.StepCompleteWhen((_runOneStep OR _runAllSteps) AND _finishStep);

    IF _runOneStep THEN
        _runOneStep := FALSE;
        RETURN;
    END_IF
END_IF

IF SUPER^.Step(919, TRUE, 'Step number 919') THEN
    SUPER^.StepCompleteWhen((_runOneStep OR _runAllSteps) AND _finishStep);

    IF _runOneStep THEN
        _runOneStep := FALSE;
        RETURN;
    END_IF
END_IF

IF SUPER^.Step(920, TRUE, 'Step number 920') THEN
    SUPER^.StepCompleteWhen((_runOneStep OR _runAllSteps) AND _finishStep);

    IF _runOneStep THEN
        _runOneStep := FALSE;
        RETURN;
    END_IF
END_IF

IF SUPER^.Step(921, TRUE, 'Step number 921') THEN
    SUPER^.StepCompleteWhen((_runOneStep OR _runAllSteps) AND _finishStep);

    IF _runOneStep THEN
        _runOneStep := FALSE;
        RETURN;
    END_IF
END_IF

IF SUPER^.Step(922, TRUE, 'Step number 922') THEN
    SUPER^.StepCompleteWhen((_runOneStep OR _runAllSteps) AND _finishStep);

    IF _runOneStep THEN
        _runOneStep := FALSE;
        RETURN;
    END_IF
END_IF

IF SUPER^.Step(923, TRUE, 'Step number 923') THEN
    SUPER^.StepCompleteWhen((_runOneStep OR _runAllSteps) AND _finishStep);

    IF _runOneStep THEN
        _runOneStep := FALSE;
        RETURN;
    END_IF
END_IF

IF SUPER^.Step(924, TRUE, 'Step number 924') THEN
    SUPER^.StepCompleteWhen((_runOneStep OR _runAllSteps) AND _finishStep);

    IF _runOneStep THEN
        _runOneStep := FALSE;
        RETURN;
    END_IF
END_IF

IF SUPER^.Step(925, TRUE, 'Step number 925') THEN
    SUPER^.StepCompleteWhen((_runOneStep OR _runAllSteps) AND _finishStep);

    IF _runOneStep THEN
        _runOneStep := FALSE;
        RETURN;
    END_IF
END_IF

IF SUPER^.Step(926, TRUE, 'Step number 926') THEN
    SUPER^.StepCompleteWhen((_runOneStep OR _runAllSteps) AND _finishStep);

    IF _runOneStep THEN
        _runOneStep := FALSE;
        RETURN;
    END_IF
END_IF

IF SUPER^.Step(927, TRUE, 'Step number 927') THEN
    SUPER^.StepCompleteWhen((_runOneStep OR _runAllSteps) AND _finishStep);

    IF _runOneStep THEN
        _runOneStep := FALSE;
        RETURN;
    END_IF
END_IF

IF SUPER^.Step(928, TRUE, 'Step number 928') THEN
    SUPER^.StepCompleteWhen((_runOneStep OR _runAllSteps) AND _finishStep);

    IF _runOneStep THEN
        _runOneStep := FALSE;
        RETURN;
    END_IF
END_IF

IF SUPER^.Step(929, TRUE, 'Step number 929') THEN
    SUPER^.StepCompleteWhen((_runOneStep OR _runAllSteps) AND _finishStep);

    IF _runOneStep THEN
        _runOneStep := FALSE;
        RETURN;
    END_IF
END_IF

IF SUPER^.Step(930, TRUE, 'Step number 930') THEN
    SUPER^.StepCompleteWhen((_runOneStep OR _runAllSteps) AND _finishStep);

    IF _runOneStep THEN
        _runOneStep := FALSE;
        RETURN;
    END_IF
END_IF

IF SUPER^.Step(931, TRUE, 'Step number 931') THEN
    SUPER^.StepCompleteWhen((_runOneStep OR _runAllSteps) AND _finishStep);

    IF _runOneStep THEN
        _runOneStep := FALSE;
        RETURN;
    END_IF
END_IF

IF SUPER^.Step(932, TRUE, 'Step number 932') THEN
    SUPER^.StepCompleteWhen((_runOneStep OR _runAllSteps) AND _finishStep);

    IF _runOneStep THEN
        _runOneStep := FALSE;
        RETURN;
    END_IF
END_IF

IF SUPER^.Step(933, TRUE, 'Step number 933') THEN
    SUPER^.StepCompleteWhen((_runOneStep OR _runAllSteps) AND _finishStep);

    IF _runOneStep THEN
        _runOneStep := FALSE;
        RETURN;
    END_IF
END_IF

IF SUPER^.Step(934, TRUE, 'Step number 934') THEN
    SUPER^.StepCompleteWhen((_runOneStep OR _runAllSteps) AND _finishStep);

    IF _runOneStep THEN
        _runOneStep := FALSE;
        RETURN;
    END_IF
END_IF

IF SUPER^.Step(935, TRUE, 'Step number 935') THEN
    SUPER^.StepCompleteWhen((_runOneStep OR _runAllSteps) AND _finishStep);

    IF _runOneStep THEN
        _runOneStep := FALSE;
        RETURN;
    END_IF
END_IF

IF SUPER^.Step(936, TRUE, 'Step number 936') THEN
    SUPER^.StepCompleteWhen((_runOneStep OR _runAllSteps) AND _finishStep);

    IF _runOneStep THEN
        _runOneStep := FALSE;
        RETURN;
    END_IF
END_IF

IF SUPER^.Step(937, TRUE, 'Step number 937') THEN
    SUPER^.StepCompleteWhen((_runOneStep OR _runAllSteps) AND _finishStep);

    IF _runOneStep THEN
        _runOneStep := FALSE;
        RETURN;
    END_IF
END_IF

IF SUPER^.Step(938, TRUE, 'Step number 938') THEN
    SUPER^.StepCompleteWhen((_runOneStep OR _runAllSteps) AND _finishStep);

    IF _runOneStep THEN
        _runOneStep := FALSE;
        RETURN;
    END_IF
END_IF

IF SUPER^.Step(939, TRUE, 'Step number 939') THEN
    SUPER^.StepCompleteWhen((_runOneStep OR _runAllSteps) AND _finishStep);

    IF _runOneStep THEN
        _runOneStep := FALSE;
        RETURN;
    END_IF
END_IF

IF SUPER^.Step(940, TRUE, 'Step number 940') THEN
    SUPER^.StepCompleteWhen((_runOneStep OR _runAllSteps) AND _finishStep);

    IF _runOneStep THEN
        _runOneStep := FALSE;
        RETURN;
    END_IF
END_IF

IF SUPER^.Step(941, TRUE, 'Step number 941') THEN
    SUPER^.StepCompleteWhen((_runOneStep OR _runAllSteps) AND _finishStep);

    IF _runOneStep THEN
        _runOneStep := FALSE;
        RETURN;
    END_IF
END_IF

IF SUPER^.Step(942, TRUE, 'Step number 942') THEN
    SUPER^.StepCompleteWhen((_runOneStep OR _runAllSteps) AND _finishStep);

    IF _runOneStep THEN
        _runOneStep := FALSE;
        RETURN;
    END_IF
END_IF

IF SUPER^.Step(943, TRUE, 'Step number 943') THEN
    SUPER^.StepCompleteWhen((_runOneStep OR _runAllSteps) AND _finishStep);

    IF _runOneStep THEN
        _runOneStep := FALSE;
        RETURN;
    END_IF
END_IF

IF SUPER^.Step(944, TRUE, 'Step number 944') THEN
    SUPER^.StepCompleteWhen((_runOneStep OR _runAllSteps) AND _finishStep);

    IF _runOneStep THEN
        _runOneStep := FALSE;
        RETURN;
    END_IF
END_IF

IF SUPER^.Step(945, TRUE, 'Step number 945') THEN
    SUPER^.StepCompleteWhen((_runOneStep OR _runAllSteps) AND _finishStep);

    IF _runOneStep THEN
        _runOneStep := FALSE;
        RETURN;
    END_IF
END_IF

IF SUPER^.Step(946, TRUE, 'Step number 946') THEN
    SUPER^.StepCompleteWhen((_runOneStep OR _runAllSteps) AND _finishStep);

    IF _runOneStep THEN
        _runOneStep := FALSE;
        RETURN;
    END_IF
END_IF

IF SUPER^.Step(947, TRUE, 'Step number 947') THEN
    SUPER^.StepCompleteWhen((_runOneStep OR _runAllSteps) AND _finishStep);

    IF _runOneStep THEN
        _runOneStep := FALSE;
        RETURN;
    END_IF
END_IF

IF SUPER^.Step(948, TRUE, 'Step number 948') THEN
    SUPER^.StepCompleteWhen((_runOneStep OR _runAllSteps) AND _finishStep);

    IF _runOneStep THEN
        _runOneStep := FALSE;
        RETURN;
    END_IF
END_IF

IF SUPER^.Step(949, TRUE, 'Step number 949') THEN
    SUPER^.StepCompleteWhen((_runOneStep OR _runAllSteps) AND _finishStep);

    IF _runOneStep THEN
        _runOneStep := FALSE;
        RETURN;
    END_IF
END_IF

IF SUPER^.Step(950, TRUE, 'Step number 950') THEN
    SUPER^.StepCompleteWhen((_runOneStep OR _runAllSteps) AND _finishStep);

    IF _runOneStep THEN
        _runOneStep := FALSE;
        RETURN;
    END_IF
END_IF

IF SUPER^.Step(951, TRUE, 'Step number 951') THEN
    SUPER^.StepCompleteWhen((_runOneStep OR _runAllSteps) AND _finishStep);

    IF _runOneStep THEN
        _runOneStep := FALSE;
        RETURN;
    END_IF
END_IF

IF SUPER^.Step(952, TRUE, 'Step number 952') THEN
    SUPER^.StepCompleteWhen((_runOneStep OR _runAllSteps) AND _finishStep);

    IF _runOneStep THEN
        _runOneStep := FALSE;
        RETURN;
    END_IF
END_IF

IF SUPER^.Step(953, TRUE, 'Step number 953') THEN
    SUPER^.StepCompleteWhen((_runOneStep OR _runAllSteps) AND _finishStep);

    IF _runOneStep THEN
        _runOneStep := FALSE;
        RETURN;
    END_IF
END_IF

IF SUPER^.Step(954, TRUE, 'Step number 954') THEN
    SUPER^.StepCompleteWhen((_runOneStep OR _runAllSteps) AND _finishStep);

    IF _runOneStep THEN
        _runOneStep := FALSE;
        RETURN;
    END_IF
END_IF

IF SUPER^.Step(955, TRUE, 'Step number 955') THEN
    SUPER^.StepCompleteWhen((_runOneStep OR _runAllSteps) AND _finishStep);

    IF _runOneStep THEN
        _runOneStep := FALSE;
        RETURN;
    END_IF
END_IF

IF SUPER^.Step(956, TRUE, 'Step number 956') THEN
    SUPER^.StepCompleteWhen((_runOneStep OR _runAllSteps) AND _finishStep);

    IF _runOneStep THEN
        _runOneStep := FALSE;
        RETURN;
    END_IF
END_IF

IF SUPER^.Step(957, TRUE, 'Step number 957') THEN
    SUPER^.StepCompleteWhen((_runOneStep OR _runAllSteps) AND _finishStep);

    IF _runOneStep THEN
        _runOneStep := FALSE;
        RETURN;
    END_IF
END_IF

IF SUPER^.Step(958, TRUE, 'Step number 958') THEN
    SUPER^.StepCompleteWhen((_runOneStep OR _runAllSteps) AND _finishStep);

    IF _runOneStep THEN
        _runOneStep := FALSE;
        RETURN;
    END_IF
END_IF

IF SUPER^.Step(959, TRUE, 'Step number 959') THEN
    SUPER^.StepCompleteWhen((_runOneStep OR _runAllSteps) AND _finishStep);

    IF _runOneStep THEN
        _runOneStep := FALSE;
        RETURN;
    END_IF
END_IF

IF SUPER^.Step(960, TRUE, 'Step number 960') THEN
    SUPER^.StepCompleteWhen((_runOneStep OR _runAllSteps) AND _finishStep);

    IF _runOneStep THEN
        _runOneStep := FALSE;
        RETURN;
    END_IF
END_IF

IF SUPER^.Step(961, TRUE, 'Step number 961') THEN
    SUPER^.StepCompleteWhen((_runOneStep OR _runAllSteps) AND _finishStep);

    IF _runOneStep THEN
        _runOneStep := FALSE;
        RETURN;
    END_IF
END_IF

IF SUPER^.Step(962, TRUE, 'Step number 962') THEN
    SUPER^.StepCompleteWhen((_runOneStep OR _runAllSteps) AND _finishStep);

    IF _runOneStep THEN
        _runOneStep := FALSE;
        RETURN;
    END_IF
END_IF

IF SUPER^.Step(963, TRUE, 'Step number 963') THEN
    SUPER^.StepCompleteWhen((_runOneStep OR _runAllSteps) AND _finishStep);

    IF _runOneStep THEN
        _runOneStep := FALSE;
        RETURN;
    END_IF
END_IF

IF SUPER^.Step(964, TRUE, 'Step number 964') THEN
    SUPER^.StepCompleteWhen((_runOneStep OR _runAllSteps) AND _finishStep);

    IF _runOneStep THEN
        _runOneStep := FALSE;
        RETURN;
    END_IF
END_IF

IF SUPER^.Step(965, TRUE, 'Step number 965') THEN
    SUPER^.StepCompleteWhen((_runOneStep OR _runAllSteps) AND _finishStep);

    IF _runOneStep THEN
        _runOneStep := FALSE;
        RETURN;
    END_IF
END_IF

IF SUPER^.Step(966, TRUE, 'Step number 966') THEN
    SUPER^.StepCompleteWhen((_runOneStep OR _runAllSteps) AND _finishStep);

    IF _runOneStep THEN
        _runOneStep := FALSE;
        RETURN;
    END_IF
END_IF

IF SUPER^.Step(967, TRUE, 'Step number 967') THEN
    SUPER^.StepCompleteWhen((_runOneStep OR _runAllSteps) AND _finishStep);

    IF _runOneStep THEN
        _runOneStep := FALSE;
        RETURN;
    END_IF
END_IF

IF SUPER^.Step(968, TRUE, 'Step number 968') THEN
    SUPER^.StepCompleteWhen((_runOneStep OR _runAllSteps) AND _finishStep);

    IF _runOneStep THEN
        _runOneStep := FALSE;
        RETURN;
    END_IF
END_IF

IF SUPER^.Step(969, TRUE, 'Step number 969') THEN
    SUPER^.StepCompleteWhen((_runOneStep OR _runAllSteps) AND _finishStep);

    IF _runOneStep THEN
        _runOneStep := FALSE;
        RETURN;
    END_IF
END_IF

IF SUPER^.Step(970, TRUE, 'Step number 970') THEN
    SUPER^.StepCompleteWhen((_runOneStep OR _runAllSteps) AND _finishStep);

    IF _runOneStep THEN
        _runOneStep := FALSE;
        RETURN;
    END_IF
END_IF

IF SUPER^.Step(971, TRUE, 'Step number 971') THEN
    SUPER^.StepCompleteWhen((_runOneStep OR _runAllSteps) AND _finishStep);

    IF _runOneStep THEN
        _runOneStep := FALSE;
        RETURN;
    END_IF
END_IF

IF SUPER^.Step(972, TRUE, 'Step number 972') THEN
    SUPER^.StepCompleteWhen((_runOneStep OR _runAllSteps) AND _finishStep);

    IF _runOneStep THEN
        _runOneStep := FALSE;
        RETURN;
    END_IF
END_IF

IF SUPER^.Step(973, TRUE, 'Step number 973') THEN
    SUPER^.StepCompleteWhen((_runOneStep OR _runAllSteps) AND _finishStep);

    IF _runOneStep THEN
        _runOneStep := FALSE;
        RETURN;
    END_IF
END_IF

IF SUPER^.Step(974, TRUE, 'Step number 974') THEN
    SUPER^.StepCompleteWhen((_runOneStep OR _runAllSteps) AND _finishStep);

    IF _runOneStep THEN
        _runOneStep := FALSE;
        RETURN;
    END_IF
END_IF

IF SUPER^.Step(975, TRUE, 'Step number 975') THEN
    SUPER^.StepCompleteWhen((_runOneStep OR _runAllSteps) AND _finishStep);

    IF _runOneStep THEN
        _runOneStep := FALSE;
        RETURN;
    END_IF
END_IF

IF SUPER^.Step(976, TRUE, 'Step number 976') THEN
    SUPER^.StepCompleteWhen((_runOneStep OR _runAllSteps) AND _finishStep);

    IF _runOneStep THEN
        _runOneStep := FALSE;
        RETURN;
    END_IF
END_IF

IF SUPER^.Step(977, TRUE, 'Step number 977') THEN
    SUPER^.StepCompleteWhen((_runOneStep OR _runAllSteps) AND _finishStep);

    IF _runOneStep THEN
        _runOneStep := FALSE;
        RETURN;
    END_IF
END_IF

IF SUPER^.Step(978, TRUE, 'Step number 978') THEN
    SUPER^.StepCompleteWhen((_runOneStep OR _runAllSteps) AND _finishStep);

    IF _runOneStep THEN
        _runOneStep := FALSE;
        RETURN;
    END_IF
END_IF

IF SUPER^.Step(979, TRUE, 'Step number 979') THEN
    SUPER^.StepCompleteWhen((_runOneStep OR _runAllSteps) AND _finishStep);

    IF _runOneStep THEN
        _runOneStep := FALSE;
        RETURN;
    END_IF
END_IF

IF SUPER^.Step(980, TRUE, 'Step number 980') THEN
    SUPER^.StepCompleteWhen((_runOneStep OR _runAllSteps) AND _finishStep);

    IF _runOneStep THEN
        _runOneStep := FALSE;
        RETURN;
    END_IF
END_IF

IF SUPER^.Step(981, TRUE, 'Step number 981') THEN
    SUPER^.StepCompleteWhen((_runOneStep OR _runAllSteps) AND _finishStep);

    IF _runOneStep THEN
        _runOneStep := FALSE;
        RETURN;
    END_IF
END_IF

IF SUPER^.Step(982, TRUE, 'Step number 982') THEN
    SUPER^.StepCompleteWhen((_runOneStep OR _runAllSteps) AND _finishStep);

    IF _runOneStep THEN
        _runOneStep := FALSE;
        RETURN;
    END_IF
END_IF

IF SUPER^.Step(983, TRUE, 'Step number 983') THEN
    SUPER^.StepCompleteWhen((_runOneStep OR _runAllSteps) AND _finishStep);

    IF _runOneStep THEN
        _runOneStep := FALSE;
        RETURN;
    END_IF
END_IF

IF SUPER^.Step(984, TRUE, 'Step number 984') THEN
    SUPER^.StepCompleteWhen((_runOneStep OR _runAllSteps) AND _finishStep);

    IF _runOneStep THEN
        _runOneStep := FALSE;
        RETURN;
    END_IF
END_IF

IF SUPER^.Step(985, TRUE, 'Step number 985') THEN
    SUPER^.StepCompleteWhen((_runOneStep OR _runAllSteps) AND _finishStep);

    IF _runOneStep THEN
        _runOneStep := FALSE;
        RETURN;
    END_IF
END_IF

IF SUPER^.Step(986, TRUE, 'Step number 986') THEN
    SUPER^.StepCompleteWhen((_runOneStep OR _runAllSteps) AND _finishStep);

    IF _runOneStep THEN
        _runOneStep := FALSE;
        RETURN;
    END_IF
END_IF

IF SUPER^.Step(987, TRUE, 'Step number 987') THEN
    SUPER^.StepCompleteWhen((_runOneStep OR _runAllSteps) AND _finishStep);

    IF _runOneStep THEN
        _runOneStep := FALSE;
        RETURN;
    END_IF
END_IF

IF SUPER^.Step(988, TRUE, 'Step number 988') THEN
    SUPER^.StepCompleteWhen((_runOneStep OR _runAllSteps) AND _finishStep);

    IF _runOneStep THEN
        _runOneStep := FALSE;
        RETURN;
    END_IF
END_IF

IF SUPER^.Step(989, TRUE, 'Step number 989') THEN
    SUPER^.StepCompleteWhen((_runOneStep OR _runAllSteps) AND _finishStep);

    IF _runOneStep THEN
        _runOneStep := FALSE;
        RETURN;
    END_IF
END_IF

IF SUPER^.Step(990, TRUE, 'Step number 990') THEN
    SUPER^.StepCompleteWhen((_runOneStep OR _runAllSteps) AND _finishStep);

    IF _runOneStep THEN
        _runOneStep := FALSE;
        RETURN;
    END_IF
END_IF

IF SUPER^.Step(991, TRUE, 'Step number 991') THEN
    SUPER^.StepCompleteWhen((_runOneStep OR _runAllSteps) AND _finishStep);

    IF _runOneStep THEN
        _runOneStep := FALSE;
        RETURN;
    END_IF
END_IF

IF SUPER^.Step(992, TRUE, 'Step number 992') THEN
    SUPER^.StepCompleteWhen((_runOneStep OR _runAllSteps) AND _finishStep);

    IF _runOneStep THEN
        _runOneStep := FALSE;
        RETURN;
    END_IF
END_IF

IF SUPER^.Step(993, TRUE, 'Step number 993') THEN
    SUPER^.StepCompleteWhen((_runOneStep OR _runAllSteps) AND _finishStep);

    IF _runOneStep THEN
        _runOneStep := FALSE;
        RETURN;
    END_IF
END_IF

IF SUPER^.Step(994, TRUE, 'Step number 994') THEN
    SUPER^.StepCompleteWhen((_runOneStep OR _runAllSteps) AND _finishStep);

    IF _runOneStep THEN
        _runOneStep := FALSE;
        RETURN;
    END_IF
END_IF

IF SUPER^.Step(995, TRUE, 'Step number 995') THEN
    SUPER^.StepCompleteWhen((_runOneStep OR _runAllSteps) AND _finishStep);

    IF _runOneStep THEN
        _runOneStep := FALSE;
        RETURN;
    END_IF
END_IF

IF SUPER^.Step(996, TRUE, 'Step number 996') THEN
    SUPER^.StepCompleteWhen((_runOneStep OR _runAllSteps) AND _finishStep);

    IF _runOneStep THEN
        _runOneStep := FALSE;
        RETURN;
    END_IF
END_IF

IF SUPER^.Step(997, TRUE, 'Step number 997') THEN
    SUPER^.StepCompleteWhen((_runOneStep OR _runAllSteps) AND _finishStep);

    IF _runOneStep THEN
        _runOneStep := FALSE;
        RETURN;
    END_IF
END_IF

IF SUPER^.Step(998, TRUE, 'Step number 998') THEN
    SUPER^.StepCompleteWhen((_runOneStep OR _runAllSteps) AND _finishStep);

    IF _runOneStep THEN
        _runOneStep := FALSE;
        RETURN;
    END_IF
END_IF

IF SUPER^.Step(999, TRUE, 'Step number 999') THEN
    SUPER^.StepCompleteWhen((_runOneStep OR _runAllSteps) AND _finishStep);

    IF _runOneStep THEN
        _runOneStep := FALSE;
        RETURN;
    END_IF
END_IF

IF SUPER^.Step(1000, TRUE, 'Step number 1000') THEN
    SUPER^.StepCompleteWhen((_runOneStep OR _runAllSteps) AND _finishStep);

    IF _runOneStep THEN
        _runOneStep := FALSE;
        RETURN;
    END_IF
END_IF

IF SUPER^.Step(1001, TRUE, 'Step number 1001') THEN
    SUPER^.StepCompleteWhen((_runOneStep OR _runAllSteps) AND _finishStep);

    IF _runOneStep THEN
        _runOneStep := FALSE;
        RETURN;
    END_IF
END_IF

IF SUPER^.Step(1002, TRUE, 'Step number 1002') THEN
    SUPER^.StepCompleteWhen((_runOneStep OR _runAllSteps) AND _finishStep);

    IF _runOneStep THEN
        _runOneStep := FALSE;
        RETURN;
    END_IF
END_IF

IF SUPER^.Step(1003, TRUE, 'Step number 1003') THEN
    SUPER^.StepCompleteWhen((_runOneStep OR _runAllSteps) AND _finishStep);

    IF _runOneStep THEN
        _runOneStep := FALSE;
        RETURN;
    END_IF
END_IF

IF SUPER^.Step(1004, TRUE, 'Step number 1004') THEN
    SUPER^.StepCompleteWhen((_runOneStep OR _runAllSteps) AND _finishStep);

    IF _runOneStep THEN
        _runOneStep := FALSE;
        RETURN;
    END_IF
END_IF

IF SUPER^.Step(1005, TRUE, 'Step number 1005') THEN
    SUPER^.StepCompleteWhen((_runOneStep OR _runAllSteps) AND _finishStep);

    IF _runOneStep THEN
        _runOneStep := FALSE;
        RETURN;
    END_IF
END_IF

IF SUPER^.Step(1006, TRUE, 'Step number 1006') THEN
    SUPER^.StepCompleteWhen((_runOneStep OR _runAllSteps) AND _finishStep);

    IF _runOneStep THEN
        _runOneStep := FALSE;
        RETURN;
    END_IF
END_IF

IF SUPER^.Step(1007, TRUE, 'Step number 1007') THEN
    SUPER^.StepCompleteWhen((_runOneStep OR _runAllSteps) AND _finishStep);

    IF _runOneStep THEN
        _runOneStep := FALSE;
        RETURN;
    END_IF
END_IF

IF SUPER^.Step(1008, TRUE, 'Step number 1008') THEN
    SUPER^.StepCompleteWhen((_runOneStep OR _runAllSteps) AND _finishStep);

    IF _runOneStep THEN
        _runOneStep := FALSE;
        RETURN;
    END_IF
END_IF

IF SUPER^.Step(1009, TRUE, 'Step number 1009') THEN
    SUPER^.StepCompleteWhen((_runOneStep OR _runAllSteps) AND _finishStep);

    IF _runOneStep THEN
        _runOneStep := FALSE;
        RETURN;
    END_IF
END_IF

IF SUPER^.Step(1010, TRUE, 'Step number 1010') THEN
    SUPER^.StepCompleteWhen((_runOneStep OR _runAllSteps) AND _finishStep);

    IF _runOneStep THEN
        _runOneStep := FALSE;
        RETURN;
    END_IF
END_IF

IF SUPER^.Step(1011, TRUE, 'Step number 1011') THEN
    SUPER^.StepCompleteWhen((_runOneStep OR _runAllSteps) AND _finishStep);

    IF _runOneStep THEN
        _runOneStep := FALSE;
        RETURN;
    END_IF
END_IF

IF SUPER^.Step(1012, TRUE, 'Step number 1012') THEN
    SUPER^.StepCompleteWhen((_runOneStep OR _runAllSteps) AND _finishStep);

    IF _runOneStep THEN
        _runOneStep := FALSE;
        RETURN;
    END_IF
END_IF

IF SUPER^.Step(1013, TRUE, 'Step number 1013') THEN
    SUPER^.StepCompleteWhen((_runOneStep OR _runAllSteps) AND _finishStep);

    IF _runOneStep THEN
        _runOneStep := FALSE;
        RETURN;
    END_IF
END_IF

IF SUPER^.Step(1014, TRUE, 'Step number 1014') THEN
    SUPER^.StepCompleteWhen((_runOneStep OR _runAllSteps) AND _finishStep);

    IF _runOneStep THEN
        _runOneStep := FALSE;
        RETURN;
    END_IF
END_IF

IF SUPER^.Step(1015, TRUE, 'Step number 1015') THEN
    SUPER^.StepCompleteWhen((_runOneStep OR _runAllSteps) AND _finishStep);

    IF _runOneStep THEN
        _runOneStep := FALSE;
        RETURN;
    END_IF
END_IF

IF SUPER^.Step(1016, TRUE, 'Step number 1016') THEN
    SUPER^.StepCompleteWhen((_runOneStep OR _runAllSteps) AND _finishStep);

    IF _runOneStep THEN
        _runOneStep := FALSE;
        RETURN;
    END_IF
END_IF

IF SUPER^.Step(1017, TRUE, 'Step number 1017') THEN
    SUPER^.StepCompleteWhen((_runOneStep OR _runAllSteps) AND _finishStep);

    IF _runOneStep THEN
        _runOneStep := FALSE;
        RETURN;
    END_IF
END_IF

IF SUPER^.Step(1018, TRUE, 'Step number 1018') THEN
    SUPER^.StepCompleteWhen((_runOneStep OR _runAllSteps) AND _finishStep);

    IF _runOneStep THEN
        _runOneStep := FALSE;
        RETURN;
    END_IF
END_IF

IF SUPER^.Step(1019, TRUE, 'Step number 1019') THEN
    SUPER^.StepCompleteWhen((_runOneStep OR _runAllSteps) AND _finishStep);

    IF _runOneStep THEN
        _runOneStep := FALSE;
        RETURN;
    END_IF
END_IF

IF SUPER^.Step(1020, TRUE, 'Step number 1020') THEN
    SUPER^.StepCompleteWhen((_runOneStep OR _runAllSteps) AND _finishStep);

    IF _runOneStep THEN
        _runOneStep := FALSE;
        RETURN;
    END_IF
END_IF

IF SUPER^.Step(1021, TRUE, 'Step number 1021') THEN
    SUPER^.StepCompleteWhen((_runOneStep OR _runAllSteps) AND _finishStep);

    IF _runOneStep THEN
        _runOneStep := FALSE;
        RETURN;
    END_IF
END_IF

IF SUPER^.Step(1022, TRUE, 'Step number 1022') THEN
    SUPER^.StepCompleteWhen((_runOneStep OR _runAllSteps) AND _finishStep);

    IF _runOneStep THEN
        _runOneStep := FALSE;
        RETURN;
    END_IF
END_IF

IF SUPER^.Step(1023, TRUE, 'Step number 1023') THEN
    SUPER^.StepCompleteWhen((_runOneStep OR _runAllSteps) AND _finishStep);

    IF _runOneStep THEN
        _runOneStep := FALSE;
        RETURN;
    END_IF
END_IF

//******************************************************************
IF SUPER^.Step(_stepId, _enabled, _stepDescription) THEN
    SUPER^.StepCompleteWhen((_runOneStep OR _runAllSteps) AND _finishStep);

    IF _runOneStep THEN
        _runOneStep := FALSE;
        RETURN;
    END_IF
END_IF
END_METHOD

METHOD PROTECTED OnSequenceCompleted
_onSequenceCompleteCount := _onSequenceCompleteCount + 1;
END_METHOD

METHOD PROTECTED OnSequencerError
VAR_INPUT
    inErrorId : eSequencerError;
END_VAR
CASE inErrorId OF
    eSequencerError.noError:
        _onSequencerErrorCount := _onSequencerErrorCount + 0;
    eSequencerError.NotUniqueStepId:
        _onSequencerErrorCount := _onSequencerErrorCount + 10;
    eSequencerError.StepIdHasBeenChanged:
        _onSequencerErrorCount := _onSequencerErrorCount + 20;
    eSequencerError.OrderOfTheStepHasBeenChanged:
        _onSequencerErrorCount := _onSequencerErrorCount + 40;
    eSequencerError.StepWithRequestedIdDoesNotExists:
        _onSequencerErrorCount := _onSequencerErrorCount + 50;
    eSequencerError.MultipleRequestStepMethodCall:
        _onSequencerErrorCount := _onSequencerErrorCount + 60;
    eSequencerError.StepIdTooLow:
        _onSequencerErrorCount := _onSequencerErrorCount + 70;
    eSequencerError.StepIdTooHigh:
        _onSequencerErrorCount := _onSequencerErrorCount + 80;
ELSE
    _onSequencerErrorCount := _onSequencerErrorCount + 0;
END_CASE
END_METHOD

METHOD PROTECTED OnStateChange
VAR_INPUT
    PreviousState : INT;
    NewState : INT;
END_VAR
THIS^._onStateChangeCount := THIS^._onStateChangeCount + 1;
_stateChangeFrom := PreviousState;
_stateChangeTo := NewState;

IF _callRestoreInOnStateChange THEN
    Restore();
END_IF
END_METHOD

METHOD PROTECTED OnStepCompleted
_onCompleteStepCount := _onCompleteStepCount + 1;
END_METHOD

PROPERTY INTERNAL RequestStepCycle : UINT
GET
RequestStepCycle := _requestStepCycle;
END_GET
SET
_requestStepCycle := RequestStepCycle;
END_SET
END_PROPERTY

METHOD INTERNAL SequencerClose
SUPER^._Close();
END_METHOD

METHOD INTERNAL SequencerHasError : BOOL
SequencerHasError := SUPER^._sequencerHasError;
END_METHOD

METHOD INTERNAL SequencerOpen
SUPER^._Open();
END_METHOD

METHOD INTERNAL SetChildState
VAR_INPUT
    inState : INT;
END_VAR
THIS^._myTcoState.ChangeState(inState);
END_METHOD

METHOD INTERNAL SetCurrentStep
VAR_INPUT
    inStepID : INT;
    inStepDescription : STRING(254);
END_VAR
THIS^._currentStep.ID := inStepID;
THIS^._currentStep.Description := inStepDescription;
END_METHOD

METHOD SetCurrentStepToErrorState : BOOL
_currentStep.Status := TcoCore.eStepStatus.Error;
SetCurrentStepToErrorState := _currentStep.Status = TcoCore.eStepStatus.Error;
END_METHOD

METHOD SetCyclicMode : BOOL
ModeController.Mode := eSequencerMode.CyclicMode;
SetCyclicMode := ModeController.Mode = eSequencerMode.CyclicMode;
END_METHOD

METHOD SetInvalidMode : BOOL
ModeController.Mode := eSequencerMode.Invalid;
SetInvalidMode := ModeController.Mode = eSequencerMode.Invalid;
END_METHOD

METHOD INTERNAL SetNumberOfSteps
VAR_INPUT
    inNumberOfSteps : UINT;
END_VAR
_stepCounter := inNumberOfSteps;
_numberOfStepsInSequence := inNumberOfSteps;
_previousNumberOfStepsInSequence := inNumberOfSteps;
END_METHOD

METHOD INTERNAL SetSequenceAsChecked
_stepIDUniquenessChecked := TRUE;
_StepIdUniquenessControlState := eStepIdUniquenessControlState.Done;
END_METHOD

METHOD INTERNAL SetSequenceAsNotChecked
_stepIDUniquenessChecked := FALSE;
_StepIdUniquenessControlState := eStepIdUniquenessControlState.NotYetStarted;
END_METHOD

METHOD SetStepMode : BOOL
ModeController.Mode := eSequencerMode.StepMode;
SetStepMode := ModeController.Mode = eSequencerMode.StepMode;
END_METHOD

METHOD INTERNAL SetTestParams
VAR_INPUT
    inRunOneStep : BOOL;
    inRunAllSteps : BOOL;
    inFinishStep : BOOL;
    inID : UINT;
    inEnabled : BOOL;
    inStepDescription : STRING(254);
END_VAR
THIS^._runOneStep := inRunOneStep;
THIS^._runAllSteps := inRunAllSteps;
THIS^._finishStep := inFinishStep;
THIS^._stepId := inID;
THIS^._enabled := inEnabled;
THIS^._stepDescription := inStepDescription;
END_METHOD

METHOD StepCount
VAR_INPUT
    inTotalStepNumber : UINT;
    inFinishStep : BOOL;
END_VAR
VAR
    i : INT;
    _lastStepId : INT;
END_VAR
FOR i := 0 TO inTotalStepNumber DO
    IF SUPER^.Step(i, TRUE, CONCAT('Step number ', INT_TO_STRING(i))) THEN
        SUPER^.StepCompleteWhen(inFinishStep);
    END_IF
END_FOR
END_METHOD

{attribute 'TcRpcEnable'}
METHOD INTERNAL UpdateCurrentStepDetails
_currentStepId := SUPER^._currentStep.ID;
_currentStepOrder := SUPER^._currentStep.Order;
_currentStepEnabled := SUPER^._currentStep.Enabled;
_currentStepDescription := SUPER^._currentStep.Description;
_currentStepStatus := SUPER^._currentStep.Status;
_currentStepDuration := SUPER^._currentStep.Duration;
END_METHOD

END_FUNCTION_BLOCK

// ---- Tests/TcoSequencer/TcoSequencerNonAutoRestorableTest.TcPOU
FUNCTION_BLOCK TcoSequencerNonAutoRestorableTest EXTENDS TcoCore._internals_TcoContext
VAR
    _callMyPlcInstance : BOOL := FALSE;
    _sequencer : _TcoSequencer(THIS^, eRestoreMode.None);
    _runPLCinstanceOnce : BOOL := FALSE;
    _runPLCinstanceCyclicaly : BOOL := FALSE;
    _stepID : INT := 32764;
    _enabled : BOOL;
    _stepDescription : STRING := 'Last step sequence message';
    _runOneStep : BOOL;
    _runAllSteps : BOOL;
    _finishStep : BOOL;
    _restore : BOOL;
    _cycleCount : INT;
    _restoreCycleCount : INT;
    _init : BOOL;
END_VAR

IF _callMyPlcInstance THEN
    IF NOT _init THEN
        ContextOpen();
        ContextClose();
        _init := THIS^._rtc.IsValid;
    END_IF

    IF _restore THEN
        ContextOpen();
        THIS^._sequencer.Restore();
        _restoreCycleCount := _restoreCycleCount + 1;
        _restore := FALSE;
        ContextClose();
        RETURN;
    END_IF

    IF _runPLCinstanceOnce AND NOT _runPLCinstanceCyclicaly THEN
        ContextOpen();
        THIS^.PLCinstanceRun(_stepID, _enabled, _stepDescription);
        _cycleCount := _cycleCount + 1;
        _runPLCinstanceOnce := FALSE;
        ContextClose();
    END_IF

    IF _runPLCinstanceCyclicaly AND NOT _runPLCinstanceOnce THEN
        ContextOpen();
        THIS^.PLCinstanceRun(_stepID, _enabled, _stepDescription);
        _cycleCount := _cycleCount + 1;
        ContextClose();
    END_IF
END_IF;

{attribute 'TcRpcEnable'}
METHOD ChildHasAutoRestoreEnabled : BOOL;
ChildHasAutoRestoreEnabled := _sequencer.ChildHasAutoRestoreEnabled();
END_METHOD

{attribute 'TcRpcEnable'}
METHOD ChildIsAutoRestorable : BOOL;
ChildIsAutoRestorable := _sequencer.ChildIsAutoRestorable();
END_METHOD

{attribute 'TcRpcEnable'}
METHOD CleanupPointers
_sequencer.CleanupPointers();
END_METHOD

{attribute 'TcRpcEnable'}
METHOD ClearNumberOfSteps
_sequencer.ClearNumberOfSteps();
END_METHOD

{attribute 'TcRpcEnable'}
METHOD PROTECTED ContextClose
SUPER^._Close();
END_METHOD

{attribute 'TcRpcEnable'}
METHOD ContextOpen
SUPER^._Open();
END_METHOD

{attribute 'TcRpcEnable'}
METHOD GetChildState : INT
GetChildState := _sequencer.GetChildState();
END_METHOD

{attribute 'TcRpcEnable'}
METHOD GetCurrentStepOrder : UINT
GetCurrentStepOrder := _sequencer._currentStep.Order;
END_METHOD

{attribute 'TcRpcEnable'}
METHOD GetNumberOfStepsInSequence : UINT
GetNumberOfStepsInSequence := _sequencer._numberOfStepsInSequence;
END_METHOD

{attribute 'TcRpcEnable'}
METHOD GetOrderOfTheCurrentlyEvaluatedStep : UINT
GetOrderOfTheCurrentlyEvaluatedStep := _sequencer._theOrderOfTheCurrentlyEvaluatedStep;
END_METHOD

{attribute 'TcRpcEnable'}
METHOD GetOrderOfTheCurrentlyExecutedStep : UINT
GetOrderOfTheCurrentlyExecutedStep := _sequencer._theOrderOfTheCurrentlyExecutedStep;
END_METHOD

{attribute 'TcRpcEnable'}
METHOD GetPreviousNumberOfStepsInSequence : UINT
GetPreviousNumberOfStepsInSequence := _sequencer._previousNumberOfStepsInSequence;
END_METHOD

{attribute 'TcRpcEnable'}
METHOD GetRequestStepCycle : UINT
GetRequestStepCycle := _sequencer.RequestStepCycle;
END_METHOD

{attribute 'TcRpcEnable'}
METHOD GetSequencerErrorId : INT
GetSequencerErrorId := _sequencer.GetSequencerErrorId();
END_METHOD

{attribute 'TcRpcEnable'}
METHOD GetTextOfTheMostImportantMessage : STRING(254)
GetTextOfTheMostImportantMessage := THIS^._sequencer.GetTextOfTheMostImportantMessage();
END_METHOD

{attribute 'TcRpcEnable'}
METHOD HasAutoRestoreEnabled : BOOL;
HasAutoRestoreEnabled := _sequencer.HasAutoRestoreEnabled();
END_METHOD

{attribute 'TcRpcEnable'}
METHOD IsAutoRestorable : BOOL;
IsAutoRestorable := _sequencer.IsAutoRestorable();
END_METHOD

{attribute 'TcRpcEnable'}
METHOD IsFirstStepEntry : BOOL
IsFirstStepEntry := THIS^._sequencer.IsFirstStepEntry();
END_METHOD

METHOD PROTECTED Main
END_METHOD

{attribute 'TcRpcEnable'}
METHOD PLCinstanceRun
VAR_INPUT
    inStepId : UINT;
    inEnabled : BOOL;
    inStepDescription : STRING(254);
END_VAR
THIS^._sequencer.SetTestParams(_runOneStep,
    _runAllSteps,
    _finishStep,
    inStepId,
    inEnabled,
    inStepDescription);

THIS^._sequencer.Run();
END_METHOD

{attribute 'TcRpcEnable'}
METHOD RequestStep
VAR_INPUT
    inRequestedStepId : INT;
END_VAR
_sequencer._RequestStep(inRequestedStepId);
END_METHOD

{attribute 'TcRpcEnable'}
METHOD Restore
_sequencer.Restore();
END_METHOD

{attribute 'TcRpcEnable'}
METHOD SequenceComplete
_sequencer._SequenceComplete();
END_METHOD

{attribute 'TcRpcEnable'}
METHOD SequencerClose
THIS^._sequencer.SequencerClose();
END_METHOD

{attribute 'TcRpcEnable'}
METHOD SequencerHasError : BOOL
SequencerHasError := _sequencer.SequencerHasError();
END_METHOD

{attribute 'TcRpcEnable'}
METHOD SequencerOpen
THIS^._sequencer.SequencerOpen();
END_METHOD

{attribute 'TcRpcEnable'}
METHOD SetChildState
VAR_INPUT
    inState : INT;
END_VAR
_sequencer.SetChildState(inState);
END_METHOD

{attribute 'TcRpcEnable'}
METHOD SetCurrentStep
VAR_INPUT
    inStepID : INT;
    inStepDescription : STRING(254);
END_VAR
_sequencer.SetCurrentStep(inStepID := inStepID, inStepDescription := inStepDescription);
END_METHOD

{attribute 'TcRpcEnable'}
METHOD SetCurrentStepToErrorState : BOOL
SetCurrentStepToErrorState := _sequencer.SetCurrentStepToErrorState();
END_METHOD

{attribute 'TcRpcEnable'}
METHOD SetCyclicMode : BOOL
SetCyclicMode := _sequencer.SetCyclicMode();
END_METHOD

{attribute 'TcRpcEnable'}
METHOD SetInvalidMode : BOOL
SetInvalidMode := _sequencer.SetInvalidMode();
END_METHOD

{attribute 'TcRpcEnable'}
METHOD SetNumberOfSteps : UINT
VAR_INPUT
    inNumberOfSteps : UINT;
END_VAR
_sequencer.SetNumberOfSteps(inNumberOfSteps);
SetNumberOfSteps := _sequencer._numberOfStepsInSequence;
END_METHOD

{attribute 'TcRpcEnable'}
METHOD SetRequestStepCycle : UINT
VAR_INPUT
    Value : UINT;
END_VAR
_sequencer.RequestStepCycle := Value;
SetRequestStepCycle := _sequencer.RequestStepCycle;
END_METHOD

{attribute 'TcRpcEnable'}
METHOD SetSequenceAsChecked : BOOL
VAR_INPUT
END_VAR
_sequencer.SetSequenceAsChecked();
END_METHOD

{attribute 'TcRpcEnable'}
METHOD SetSequenceAsNotChecked : BOOL
VAR_INPUT
END_VAR
_sequencer.SetSequenceAsNotChecked();
END_METHOD

{attribute 'TcRpcEnable'}
METHOD SetStepMode : BOOL
SetStepMode := _sequencer.SetStepMode();
END_METHOD

{attribute 'TcRpcEnable'}
METHOD Step : BOOL
VAR_INPUT
    inStepId : INT;
    inEnabled : BOOL;
    inStepDescription : STRING(254);
END_VAR
Step := _sequencer._Step(inStepID := inStepId, inEnabled := inEnabled, inStepDescription := inStepDescription);
END_METHOD

{attribute 'TcRpcEnable'}
METHOD StepBackward
_sequencer._StepBackward();
END_METHOD

{attribute 'TcRpcEnable'}
METHOD StepCompleteWhen
VAR_INPUT
    inCondition : BOOL;
END_VAR
_sequencer._StepCompleteWhen(inCondition);
END_METHOD

{attribute 'TcRpcEnable'}
METHOD StepForward
_sequencer._StepForward();
END_METHOD

{attribute 'TcRpcEnable'}
METHOD StepIn
_sequencer._StepIn();
END_METHOD

{attribute 'TcRpcEnable'}
METHOD UpdateCurrentStepDetails
VAR_INPUT
END_VAR
_sequencer.UpdateCurrentStepDetails();
END_METHOD

END_FUNCTION_BLOCK

// ---- Tests/TcoSequence/TcoSequenceAutoRestorableTest.TcPOU
FUNCTION_BLOCK TcoSequenceAutoRestorableTest EXTENDS TcoCore._internals_TcoContext
VAR
    _callMyPlcInstance : BOOL := FALSE;
    _sequencer : _TcoSequence(THIS^, eRestoreMode.AutoRestoreMembers);
    _runPLCinstanceOnce : BOOL := FALSE;
    _runPLCinstanceCyclicaly : BOOL := FALSE;
    _stepID : INT := 32764;
    _enabled : BOOL;
    _stepDescription : STRING := 'Last step sequence message';
    _runOneStep : BOOL;
    _runAllSteps : BOOL;
    _finishStep : BOOL;
    _restore : BOOL;
    _cycleCount : INT;
    _restoreCycleCount : INT;
    _init : BOOL;
    _setCurrentStepPropTestData : TcoCore.StepDetails;
END_VAR

IF _callMyPlcInstance THEN
    IF NOT _init THEN
        ContextOpen();
        ContextClose();
        _init := THIS^._rtc.IsValid;
    END_IF

    IF _restore THEN
        ContextOpen();
        THIS^._sequencer.Restore();
        _restoreCycleCount := _restoreCycleCount + 1;
        _restore := FALSE;
        ContextClose();
        RETURN;
    END_IF

    IF _runPLCinstanceOnce AND NOT _runPLCinstanceCyclicaly THEN
        ContextOpen();
        THIS^.PLCinstanceRun(_stepID, _enabled, _stepDescription);
        _cycleCount := _cycleCount + 1;
        _runPLCinstanceOnce := FALSE;
        ContextClose();
    END_IF

    IF _runPLCinstanceCyclicaly AND NOT _runPLCinstanceOnce THEN
        ContextOpen();
        THIS^.PLCinstanceRun(_stepID, _enabled, _stepDescription);
        _cycleCount := _cycleCount + 1;
        ContextClose();
    END_IF
END_IF;

{attribute 'TcRpcEnable'}
METHOD ChildHasAutoRestoreEnabled : BOOL;
ChildHasAutoRestoreEnabled := _sequencer.ChildHasAutoRestoreEnabled();
END_METHOD

{attribute 'TcRpcEnable'}
METHOD ChildIsAutoRestorable : BOOL;
ChildIsAutoRestorable := _sequencer.ChildIsAutoRestorable();
END_METHOD

{attribute 'TcRpcEnable'}
METHOD CleanupPointers
_sequencer.CleanupPointers();
END_METHOD

{attribute 'TcRpcEnable'}
METHOD ClearNumberOfSteps
_sequencer.ClearNumberOfSteps();
END_METHOD

{attribute 'TcRpcEnable'}
METHOD PROTECTED ContextClose
SUPER^._Close();
END_METHOD

{attribute 'TcRpcEnable'}
METHOD ContextOpen
SUPER^._Open();
END_METHOD

{attribute 'TcRpcEnable'}
METHOD GetChildState : INT
GetChildState := _sequencer.GetChildState();
END_METHOD

{attribute 'TcRpcEnable'}
METHOD GetCurrentStepOrder : UINT
GetCurrentStepOrder := _sequencer._currentStep.Order;
END_METHOD

{attribute 'TcRpcEnable'}
METHOD GetCurrentStepPropTest
_setCurrentStepPropTestData := THIS^._sequencer.CurrentStep;
END_METHOD

{attribute 'TcRpcEnable'}
METHOD GetNumberOfStepsInSequence : UINT
GetNumberOfStepsInSequence := _sequencer._numberOfStepsInSequence;
END_METHOD

{attribute 'TcRpcEnable'}
METHOD GetOrderOfTheCurrentlyEvaluatedStep : UINT
GetOrderOfTheCurrentlyEvaluatedStep := _sequencer._theOrderOfTheCurrentlyEvaluatedStep;
END_METHOD

{attribute 'TcRpcEnable'}
METHOD GetOrderOfTheCurrentlyExecutedStep : UINT
GetOrderOfTheCurrentlyExecutedStep := _sequencer._theOrderOfTheCurrentlyExecutedStep;
END_METHOD

{attribute 'TcRpcEnable'}
METHOD GetPreviousNumberOfStepsInSequence : UINT
GetPreviousNumberOfStepsInSequence := _sequencer._previousNumberOfStepsInSequence;
END_METHOD

{attribute 'TcRpcEnable'}
METHOD GetRequestStepCycle : UINT
GetRequestStepCycle := _sequencer.RequestStepCycle;
END_METHOD

{attribute 'TcRpcEnable'}
METHOD GetSequencerErrorId : INT
GetSequencerErrorId := _sequencer.GetSequencerErrorId();
END_METHOD

{attribute 'TcRpcEnable'}
METHOD GetTextOfTheMostImportantMessage : STRING(254)
GetTextOfTheMostImportantMessage := THIS^._sequencer.GetTextOfTheMostImportantMessage();
END_METHOD

{attribute 'TcRpcEnable'}
METHOD HasAutoRestoreEnabled : BOOL;
HasAutoRestoreEnabled := _sequencer.HasAutoRestoreEnabled();
END_METHOD

{attribute 'TcRpcEnable'}
METHOD IsAutoRestorable : BOOL;
IsAutoRestorable := _sequencer.IsAutoRestorable();
END_METHOD

{attribute 'TcRpcEnable'}
METHOD IsFirstStepEntry : BOOL
IsFirstStepEntry := THIS^._sequencer.IsFirstStepEntry();
END_METHOD

METHOD PROTECTED Main
END_METHOD

{attribute 'TcRpcEnable'}
METHOD PLCinstanceRun
VAR_INPUT
    inStepId : UINT;
    inEnabled : BOOL;
    inStepDescription : STRING(254);
END_VAR
THIS^._sequencer.SetTestParams(_runOneStep,
    _runAllSteps,
    _finishStep,
    inStepId,
    inEnabled,
    inStepDescription);

THIS^._sequencer._RunExecutionSubstitute();
END_METHOD

{attribute 'TcRpcEnable'}
METHOD RequestStep
VAR_INPUT
    inRequestedStepId : INT;
END_VAR
_sequencer._RequestStep(inRequestedStepId);
END_METHOD

{attribute 'TcRpcEnable'}
METHOD Restore
_sequencer.Restore();
END_METHOD

{attribute 'TcRpcEnable'}
METHOD SequenceComplete
_sequencer._SequenceComplete();
END_METHOD

{attribute 'TcRpcEnable'}
METHOD SequencerClose
THIS^._sequencer.SequencerClose();
END_METHOD

{attribute 'TcRpcEnable'}
METHOD SequencerHasError : BOOL
SequencerHasError := _sequencer.SequencerHasError();
END_METHOD

{attribute 'TcRpcEnable'}
METHOD SequencerOpen
THIS^._sequencer.SequencerOpen();
END_METHOD

{attribute 'TcRpcEnable'}
METHOD SetChildState
VAR_INPUT
    inState : INT;
END_VAR
_sequencer.SetChildState(inState);
END_METHOD

{attribute 'TcRpcEnable'}
METHOD SetCurrentStep
VAR_INPUT
    inStepID : INT;
    inStepDescription : STRING(254);
END_VAR
_sequencer.SetCurrentStep(inStepID := inStepID, inStepDescription := inStepDescription);
END_METHOD

{attribute 'TcRpcEnable'}
METHOD SetCurrentStepToErrorState : BOOL
SetCurrentStepToErrorState := _sequencer.SetCurrentStepToErrorState();
END_METHOD

{attribute 'TcRpcEnable'}
METHOD SetCyclicMode : BOOL
SetCyclicMode := _sequencer.SetCyclicMode();
END_METHOD

{attribute 'TcRpcEnable'}
METHOD SetInvalidMode : BOOL
SetInvalidMode := _sequencer.SetInvalidMode();
END_METHOD

{attribute 'TcRpcEnable'}
METHOD SetNumberOfSteps : UINT
VAR_INPUT
    inNumberOfSteps : UINT;
END_VAR
_sequencer.SetNumberOfSteps(inNumberOfSteps);
SetNumberOfSteps := _sequencer._numberOfStepsInSequence;
END_METHOD

{attribute 'TcRpcEnable'}
METHOD SetRequestStepCycle : UINT
VAR_INPUT
    Value : UINT;
END_VAR
_sequencer.RequestStepCycle := Value;
SetRequestStepCycle := _sequencer.RequestStepCycle;
END_METHOD

{attribute 'TcRpcEnable'}
METHOD SetSequenceAsChecked : BOOL
VAR_INPUT
END_VAR
_sequencer.SetSequenceAsChecked();
END_METHOD

{attribute 'TcRpcEnable'}
METHOD SetSequenceAsNotChecked : BOOL
VAR_INPUT
END_VAR
_sequencer.SetSequenceAsNotChecked();
END_METHOD

{attribute 'TcRpcEnable'}
METHOD SetStepMode : BOOL
SetStepMode := _sequencer.SetStepMode();
END_METHOD

{attribute 'TcRpcEnable'}
METHOD Step : BOOL
VAR_INPUT
    inStepId : INT;
    inEnabled : BOOL;
    inStepDescription : STRING(254);
END_VAR
Step := _sequencer._Step(inStepID := inStepId, inEnabled := inEnabled, inStepDescription := inStepDescription);
END_METHOD

{attribute 'TcRpcEnable'}
METHOD StepBackward
_sequencer._StepBackward();
END_METHOD

{attribute 'TcRpcEnable'}
METHOD StepCompleteWhen
VAR_INPUT
    inCondition : BOOL;
END_VAR
_sequencer._StepCompleteWhen(inCondition);
END_METHOD

{attribute 'TcRpcEnable'}
METHOD StepForward
_sequencer._StepForward();
END_METHOD

{attribute 'TcRpcEnable'}
METHOD StepIn
_sequencer._StepIn();
END_METHOD

{attribute 'TcRpcEnable'}
METHOD UpdateCurrentStepDetails
VAR_INPUT
END_VAR
_sequencer.UpdateCurrentStepDetails();
END_METHOD

END_FUNCTION_BLOCK

// ---- Tests/TcoSequence/_TcoSequence.TcPOU
FUNCTION_BLOCK _TcoSequence EXTENDS TcoCore._internals_TcoSequence
VAR
    _runOneStep : BOOL;
    _runAllSteps : BOOL;
    _finishStep : BOOL;
    _stepId : INT;
    _enabled : BOOL;
    _stepDescription : STRING(254);
    _currentStepId : INT;
    _currentStepOrder : UINT;
    _currentStepEnabled : BOOL;
    _currentStepDescription : STRING(254);
    _currentStepStatus : INT;
    _currentStepDuration : TIME;
    _myTcoState : TcoState(THIS^, eRestoreMode.None);
    _onCompleteStepCount : INT;
    _onSequenceCompleteCount : INT;
    _onSequencerErrorCount : ULINT;
    _onStateChangeCount : ULINT;
    _stateChangeFrom : INT;
    _stateChangeTo : INT;
    _callRestoreInOnStateChange : BOOL;
END_VAR

METHOD _RequestStep
VAR_INPUT
    inRequestedStepId : INT;
END_VAR
THIS^.RequestStep(inRequestedStepId);
END_METHOD

METHOD _RunExecutionSubstitute
VAR_INPUT
END_VAR
THIS^.Open();
THIS^.Main();
THIS^.Close();
END_METHOD

METHOD _SequenceComplete
THIS^.CompleteSequence();
END_METHOD

METHOD INTERNAL _Step : BOOL
VAR_INPUT
    inStepId : INT;
    inEnabled : BOOL;
    inStepDescription : STRING(254);
END_VAR
_Step := SUPER^.Step(inStepID := inStepId, inEnabled := inEnabled, inStepDescription := inStepDescription);
END_METHOD

METHOD _StepBackward
THIS^.ModeController.StepBackward();
END_METHOD

METHOD _StepCompleteWhen
VAR_INPUT
    inCondition : BOOL;
END_VAR
THIS^.StepCompleteWhen(inCondition);
END_METHOD

METHOD _StepForward
THIS^.ModeController.StepForward();
END_METHOD

METHOD INTERNAL _StepIn
THIS^.ModeController.StepIn();
END_METHOD

METHOD INTERNAL ChildHasAutoRestoreEnabled : BOOL
ChildHasAutoRestoreEnabled := THIS^._myTcoState.IsAutoRestoreEnabled;
END_METHOD

METHOD INTERNAL ChildIsAutoRestorable : BOOL
ChildIsAutoRestorable := THIS^._myTcoState.AutoRestorable;
END_METHOD

METHOD INTERNAL CleanupPointers
IF (_pPreviusSteps <> 0) THEN
    __DELETE(_pPreviusSteps);
END_IF
END_METHOD

METHOD INTERNAL ClearNumberOfSteps
_stepCounter := 0;
_numberOfStepsInSequence := 0;
_previousNumberOfStepsInSequence := 0;
END_METHOD

METHOD INTERNAL GetChildState : INT
GetChildState := THIS^._myTcoState.State;
END_METHOD

{attribute 'TcRpcEnable'}
METHOD GetNumberOfStepsInSequence : UINT
GetNumberOfStepsInSequence := THIS^._numberOfStepsInSequence;
END_METHOD

METHOD INTERNAL GetSequencerErrorId : INT
GetSequencerErrorId := SUPER^._sequencerErrorId;
END_METHOD

METHOD INTERNAL GetTextOfTheMostImportantMessage : STRING(254)
GetTextOfTheMostImportantMessage := THIS^._messenger._mime.Text;
END_METHOD

METHOD INTERNAL HasAutoRestoreEnabled : BOOL
HasAutoRestoreEnabled := SUPER^.IsAutoRestoreEnabled;
END_METHOD

METHOD INTERNAL IsAutoRestorable : BOOL
IsAutoRestorable := SUPER^.AutoRestorable;
END_METHOD

METHOD INTERNAL IsFirstStepEntry : BOOL
IsFirstStepEntry := _isFirstStepEntry;
END_METHOD

METHOD PROTECTED Main : BOOL
//******************************************************************
IF SUPER^.Step(0, TRUE, 'Step number 0') THEN
    SUPER^.StepCompleteWhen((_runOneStep OR _runAllSteps) AND _finishStep);

    IF _runOneStep THEN
        _runOneStep := FALSE;
        RETURN;
    END_IF
END_IF

IF SUPER^.Step(1, TRUE, 'Step number 1') THEN
    SUPER^.StepCompleteWhen((_runOneStep OR _runAllSteps) AND _finishStep);

    IF _runOneStep THEN
        _runOneStep := FALSE;
        RETURN;
    END_IF
END_IF

IF SUPER^.Step(2, TRUE, 'Step number 2') THEN
    SUPER^.StepCompleteWhen((_runOneStep OR _runAllSteps) AND _finishStep);

    IF _runOneStep THEN
        _runOneStep := FALSE;
        RETURN;
    END_IF
END_IF

IF SUPER^.Step(3, TRUE, 'Step number 3') THEN
    SUPER^.StepCompleteWhen((_runOneStep OR _runAllSteps) AND _finishStep);

    IF _runOneStep THEN
        _runOneStep := FALSE;
        RETURN;
    END_IF
END_IF

IF SUPER^.Step(4, TRUE, 'Step number 4') THEN
    SUPER^.StepCompleteWhen((_runOneStep OR _runAllSteps) AND _finishStep);

    IF _runOneStep THEN
        _runOneStep := FALSE;
        RETURN;
    END_IF
END_IF

IF SUPER^.Step(5, TRUE, 'Step number 5') THEN
    SUPER^.StepCompleteWhen((_runOneStep OR _runAllSteps) AND _finishStep);

    IF _runOneStep THEN
        _runOneStep := FALSE;
        RETURN;
    END_IF
END_IF

IF SUPER^.Step(6, TRUE, 'Step number 6') THEN
    SUPER^.StepCompleteWhen((_runOneStep OR _runAllSteps) AND _finishStep);

    IF _runOneStep THEN
        _runOneStep := FALSE;
        RETURN;
    END_IF
END_IF

IF SUPER^.Step(7, TRUE, 'Step number 7') THEN
    SUPER^.StepCompleteWhen((_runOneStep OR _runAllSteps) AND _finishStep);

    IF _runOneStep THEN
        _runOneStep := FALSE;
        RETURN;
    END_IF
END_IF

IF SUPER^.Step(8, TRUE, 'Step number 8') THEN
    SUPER^.StepCompleteWhen((_runOneStep OR _runAllSteps) AND _finishStep);

    IF _runOneStep THEN
        _runOneStep := FALSE;
        RETURN;
    END_IF
END_IF

IF SUPER^.Step(9, TRUE, 'Step number 9') THEN
    SUPER^.StepCompleteWhen((_runOneStep OR _runAllSteps) AND _finishStep);

    IF _runOneStep THEN
        _runOneStep := FALSE;
        RETURN;
    END_IF
END_IF

IF SUPER^.Step(10, TRUE, 'Step number 10') THEN
    SUPER^.StepCompleteWhen((_runOneStep OR _runAllSteps) AND _finishStep);

    IF _runOneStep THEN
        _runOneStep := FALSE;
        RETURN;
    END_IF
END_IF

IF SUPER^.Step(11, TRUE, 'Step number 11') THEN
    SUPER^.StepCompleteWhen((_runOneStep OR _runAllSteps) AND _finishStep);

    IF _runOneStep THEN
        _runOneStep := FALSE;
        RETURN;
    END_IF
END_IF

IF SUPER^.Step(12, TRUE, 'Step number 12') THEN
    SUPER^.StepCompleteWhen((_runOneStep OR _runAllSteps) AND _finishStep);

    IF _runOneStep THEN
        _runOneStep := FALSE;
        RETURN;
    END_IF
END_IF

IF SUPER^.Step(13, TRUE, 'Step number 13') THEN
    SUPER^.StepCompleteWhen((_runOneStep OR _runAllSteps) AND _finishStep);

    IF _runOneStep THEN
        _runOneStep := FALSE;
        RETURN;
    END_IF
END_IF

IF SUPER^.Step(14, TRUE, 'Step number 14') THEN
    SUPER^.StepCompleteWhen((_runOneStep OR _runAllSteps) AND _finishStep);

    IF _runOneStep THEN
        _runOneStep := FALSE;
        RETURN;
    END_IF
END_IF

IF SUPER^.Step(15, TRUE, 'Step number 15') THEN
    SUPER^.StepCompleteWhen((_runOneStep OR _runAllSteps) AND _finishStep);

    IF _runOneStep THEN
        _runOneStep := FALSE;
        RETURN;
    END_IF
END_IF

IF SUPER^.Step(16, TRUE, 'Step number 16') THEN
    SUPER^.StepCompleteWhen((_runOneStep OR _runAllSteps) AND _finishStep);

    IF _runOneStep THEN
        _runOneStep := FALSE;
        RETURN;
    END_IF
END_IF

IF SUPER^.Step(17, TRUE, 'Step number 17') THEN
    SUPER^.StepCompleteWhen((_runOneStep OR _runAllSteps) AND _finishStep);

    IF _runOneStep THEN
        _runOneStep := FALSE;
        RETURN;
    END_IF
END_IF

IF SUPER^.Step(18, TRUE, 'Step number 18') THEN
    SUPER^.StepCompleteWhen((_runOneStep OR _runAllSteps) AND _finishStep);

    IF _runOneStep THEN
        _runOneStep := FALSE;
        RETURN;
    END_IF
END_IF

IF SUPER^.Step(19, TRUE, 'Step number 19') THEN
    SUPER^.StepCompleteWhen((_runOneStep OR _runAllSteps) AND _finishStep);

    IF _runOneStep THEN
        _runOneStep := FALSE;
        RETURN;
    END_IF
END_IF

IF SUPER^.Step(20, TRUE, 'Step number 20') THEN
    SUPER^.StepCompleteWhen((_runOneStep OR _runAllSteps) AND _finishStep);

    IF _runOneStep THEN
        _runOneStep := FALSE;
        RETURN;
    END_IF
END_IF

IF SUPER^.Step(21, TRUE, 'Step number 21') THEN
    SUPER^.StepCompleteWhen((_runOneStep OR _runAllSteps) AND _finishStep);

    IF _runOneStep THEN
        _runOneStep := FALSE;
        RETURN;
    END_IF
END_IF

IF SUPER^.Step(22, TRUE, 'Step number 22') THEN
    SUPER^.StepCompleteWhen((_runOneStep OR _runAllSteps) AND _finishStep);

    IF _runOneStep THEN
        _runOneStep := FALSE;
        RETURN;
    END_IF
END_IF

IF SUPER^.Step(23, TRUE, 'Step number 23') THEN
    SUPER^.StepCompleteWhen((_runOneStep OR _runAllSteps) AND _finishStep);

    IF _runOneStep THEN
        _runOneStep := FALSE;
        RETURN;
    END_IF
END_IF

IF SUPER^.Step(24, TRUE, 'Step number 24') THEN
    SUPER^.StepCompleteWhen((_runOneStep OR _runAllSteps) AND _finishStep);

    IF _runOneStep THEN
        _runOneStep := FALSE;
        RETURN;
    END_IF
END_IF

IF SUPER^.Step(25, TRUE, 'Step number 25') THEN
    SUPER^.StepCompleteWhen((_runOneStep OR _runAllSteps) AND _finishStep);

    IF _runOneStep THEN
        _runOneStep := FALSE;
        RETURN;
    END_IF
END_IF

IF SUPER^.Step(26, TRUE, 'Step number 26') THEN
    SUPER^.StepCompleteWhen((_runOneStep OR _runAllSteps) AND _finishStep);

    IF _runOneStep THEN
        _runOneStep := FALSE;
        RETURN;
    END_IF
END_IF

IF SUPER^.Step(27, TRUE, 'Step number 27') THEN
    SUPER^.StepCompleteWhen((_runOneStep OR _runAllSteps) AND _finishStep);

    IF _runOneStep THEN
        _runOneStep := FALSE;
        RETURN;
    END_IF
END_IF

IF SUPER^.Step(28, TRUE, 'Step number 28') THEN
    SUPER^.StepCompleteWhen((_runOneStep OR _runAllSteps) AND _finishStep);

    IF _runOneStep THEN
        _runOneStep := FALSE;
        RETURN;
    END_IF
END_IF

IF SUPER^.Step(29, TRUE, 'Step number 29') THEN
    SUPER^.StepCompleteWhen((_runOneStep OR _runAllSteps) AND _finishStep);

    IF _runOneStep THEN
        _runOneStep := FALSE;
        RETURN;
    END_IF
END_IF

IF SUPER^.Step(30, TRUE, 'Step number 30') THEN
    SUPER^.StepCompleteWhen((_runOneStep OR _runAllSteps) AND _finishStep);

    IF _runOneStep THEN
        _runOneStep := FALSE;
        RETURN;
    END_IF
END_IF

IF SUPER^.Step(31, TRUE, 'Step number 31') THEN
    SUPER^.StepCompleteWhen((_runOneStep OR _runAllSteps) AND _finishStep);

    IF _runOneStep THEN
        _runOneStep := FALSE;
        RETURN;
    END_IF
END_IF

IF SUPER^.Step(32, TRUE, 'Step number 32') THEN
    SUPER^.StepCompleteWhen((_runOneStep OR _runAllSteps) AND _finishStep);

    IF _runOneStep THEN
        _runOneStep := FALSE;
        RETURN;
    END_IF
END_IF

IF SUPER^.Step(33, TRUE, 'Step number 33') THEN
    SUPER^.StepCompleteWhen((_runOneStep OR _runAllSteps) AND _finishStep);

    IF _runOneStep THEN
        _runOneStep := FALSE;
        RETURN;
    END_IF
END_IF

IF SUPER^.Step(34, TRUE, 'Step number 34') THEN
    SUPER^.StepCompleteWhen((_runOneStep OR _runAllSteps) AND _finishStep);

    IF _runOneStep THEN
        _runOneStep := FALSE;
        RETURN;
    END_IF
END_IF

IF SUPER^.Step(35, TRUE, 'Step number 35') THEN
    SUPER^.StepCompleteWhen((_runOneStep OR _runAllSteps) AND _finishStep);

    IF _runOneStep THEN
        _runOneStep := FALSE;
        RETURN;
    END_IF
END_IF

IF SUPER^.Step(36, TRUE, 'Step number 36') THEN
    SUPER^.StepCompleteWhen((_runOneStep OR _runAllSteps) AND _finishStep);

    IF _runOneStep THEN
        _runOneStep := FALSE;
        RETURN;
    END_IF
END_IF

IF SUPER^.Step(37, TRUE, 'Step number 37') THEN
    SUPER^.StepCompleteWhen((_runOneStep OR _runAllSteps) AND _finishStep);

    IF _runOneStep THEN
        _runOneStep := FALSE;
        RETURN;
    END_IF
END_IF

IF SUPER^.Step(38, TRUE, 'Step number 38') THEN
    SUPER^.StepCompleteWhen((_runOneStep OR _runAllSteps) AND _finishStep);

    IF _runOneStep THEN
        _runOneStep := FALSE;
        RETURN;
    END_IF
END_IF

IF SUPER^.Step(39, TRUE, 'Step number 39') THEN
    SUPER^.StepCompleteWhen((_runOneStep OR _runAllSteps) AND _finishStep);

    IF _runOneStep THEN
        _runOneStep := FALSE;
        RETURN;
    END_IF
END_IF

IF SUPER^.Step(40, TRUE, 'Step number 40') THEN
    SUPER^.StepCompleteWhen((_runOneStep OR _runAllSteps) AND _finishStep);

    IF _runOneStep THEN
        _runOneStep := FALSE;
        RETURN;
    END_IF
END_IF

IF SUPER^.Step(41, TRUE, 'Step number 41') THEN
    SUPER^.StepCompleteWhen((_runOneStep OR _runAllSteps) AND _finishStep);

    IF _runOneStep THEN
        _runOneStep := FALSE;
        RETURN;
    END_IF
END_IF

IF SUPER^.Step(42, TRUE, 'Step number 42') THEN
    SUPER^.StepCompleteWhen((_runOneStep OR _runAllSteps) AND _finishStep);

    IF _runOneStep THEN
        _runOneStep := FALSE;
        RETURN;
    END_IF
END_IF

IF SUPER^.Step(43, TRUE, 'Step number 43') THEN
    SUPER^.StepCompleteWhen((_runOneStep OR _runAllSteps) AND _finishStep);

    IF _runOneStep THEN
        _runOneStep := FALSE;
        RETURN;
    END_IF
END_IF

IF SUPER^.Step(44, TRUE, 'Step number 44') THEN
    SUPER^.StepCompleteWhen((_runOneStep OR _runAllSteps) AND _finishStep);

    IF _runOneStep THEN
        _runOneStep := FALSE;
        RETURN;
    END_IF
END_IF

IF SUPER^.Step(45, TRUE, 'Step number 45') THEN
    SUPER^.StepCompleteWhen((_runOneStep OR _runAllSteps) AND _finishStep);

    IF _runOneStep THEN
        _runOneStep := FALSE;
        RETURN;
    END_IF
END_IF

IF SUPER^.Step(46, TRUE, 'Step number 46') THEN
    SUPER^.StepCompleteWhen((_runOneStep OR _runAllSteps) AND _finishStep);

    IF _runOneStep THEN
        _runOneStep := FALSE;
        RETURN;
    END_IF
END_IF

IF SUPER^.Step(47, TRUE, 'Step number 47') THEN
    SUPER^.StepCompleteWhen((_runOneStep OR _runAllSteps) AND _finishStep);

    IF _runOneStep THEN
        _runOneStep := FALSE;
        RETURN;
    END_IF
END_IF

IF SUPER^.Step(48, TRUE, 'Step number 48') THEN
    SUPER^.StepCompleteWhen((_runOneStep OR _runAllSteps) AND _finishStep);

    IF _runOneStep THEN
        _runOneStep := FALSE;
        RETURN;
    END_IF
END_IF

IF SUPER^.Step(49, TRUE, 'Step number 49') THEN
    SUPER^.StepCompleteWhen((_runOneStep OR _runAllSteps) AND _finishStep);

    IF _runOneStep THEN
        _runOneStep := FALSE;
        RETURN;
    END_IF
END_IF

IF SUPER^.Step(50, TRUE, 'Step number 50') THEN
    SUPER^.StepCompleteWhen((_runOneStep OR _runAllSteps) AND _finishStep);

    IF _runOneStep THEN
        _runOneStep := FALSE;
        RETURN;
    END_IF
END_IF

IF SUPER^.Step(51, TRUE, 'Step number 51') THEN
    SUPER^.StepCompleteWhen((_runOneStep OR _runAllSteps) AND _finishStep);

    IF _runOneStep THEN
        _runOneStep := FALSE;
        RETURN;
    END_IF
END_IF

IF SUPER^.Step(52, TRUE, 'Step number 52') THEN
    SUPER^.StepCompleteWhen((_runOneStep OR _runAllSteps) AND _finishStep);

    IF _runOneStep THEN
        _runOneStep := FALSE;
        RETURN;
    END_IF
END_IF

IF SUPER^.Step(53, TRUE, 'Step number 53') THEN
    SUPER^.StepCompleteWhen((_runOneStep OR _runAllSteps) AND _finishStep);

    IF _runOneStep THEN
        _runOneStep := FALSE;
        RETURN;
    END_IF
END_IF

IF SUPER^.Step(54, TRUE, 'Step number 54') THEN
    SUPER^.StepCompleteWhen((_runOneStep OR _runAllSteps) AND _finishStep);

    IF _runOneStep THEN
        _runOneStep := FALSE;
        RETURN;
    END_IF
END_IF

IF SUPER^.Step(55, TRUE, 'Step number 55') THEN
    SUPER^.StepCompleteWhen((_runOneStep OR _runAllSteps) AND _finishStep);

    IF _runOneStep THEN
        _runOneStep := FALSE;
        RETURN;
    END_IF
END_IF

IF SUPER^.Step(56, TRUE, 'Step number 56') THEN
    SUPER^.StepCompleteWhen((_runOneStep OR _runAllSteps) AND _finishStep);

    IF _runOneStep THEN
        _runOneStep := FALSE;
        RETURN;
    END_IF
END_IF

IF SUPER^.Step(57, TRUE, 'Step number 57') THEN
    SUPER^.StepCompleteWhen((_runOneStep OR _runAllSteps) AND _finishStep);

    IF _runOneStep THEN
        _runOneStep := FALSE;
        RETURN;
    END_IF
END_IF

IF SUPER^.Step(58, TRUE, 'Step number 58') THEN
    SUPER^.StepCompleteWhen((_runOneStep OR _runAllSteps) AND _finishStep);

    IF _runOneStep THEN
        _runOneStep := FALSE;
        RETURN;
    END_IF
END_IF

IF SUPER^.Step(59, TRUE, 'Step number 59') THEN
    SUPER^.StepCompleteWhen((_runOneStep OR _runAllSteps) AND _finishStep);

    IF _runOneStep THEN
        _runOneStep := FALSE;
        RETURN;
    END_IF
END_IF

IF SUPER^.Step(60, TRUE, 'Step number 60') THEN
    SUPER^.StepCompleteWhen((_runOneStep OR _runAllSteps) AND _finishStep);

    IF _runOneStep THEN
        _runOneStep := FALSE;
        RETURN;
    END_IF
END_IF

IF SUPER^.Step(61, TRUE, 'Step number 61') THEN
    SUPER^.StepCompleteWhen((_runOneStep OR _runAllSteps) AND _finishStep);

    IF _runOneStep THEN
        _runOneStep := FALSE;
        RETURN;
    END_IF
END_IF

IF SUPER^.Step(62, TRUE, 'Step number 62') THEN
    SUPER^.StepCompleteWhen((_runOneStep OR _runAllSteps) AND _finishStep);

    IF _runOneStep THEN
        _runOneStep := FALSE;
        RETURN;
    END_IF
END_IF

IF SUPER^.Step(63, TRUE, 'Step number 63') THEN
    SUPER^.StepCompleteWhen((_runOneStep OR _runAllSteps) AND _finishStep);

    IF _runOneStep THEN
        _runOneStep := FALSE;
        RETURN;
    END_IF
END_IF

IF SUPER^.Step(64, TRUE, 'Step number 64') THEN
    SUPER^.StepCompleteWhen((_runOneStep OR _runAllSteps) AND _finishStep);

    IF _runOneStep THEN
        _runOneStep := FALSE;
        RETURN;
    END_IF
END_IF

IF SUPER^.Step(65, TRUE, 'Step number 65') THEN
    SUPER^.StepCompleteWhen((_runOneStep OR _runAllSteps) AND _finishStep);

    IF _runOneStep THEN
        _runOneStep := FALSE;
        RETURN;
    END_IF
END_IF

IF SUPER^.Step(66, TRUE, 'Step number 66') THEN
    SUPER^.StepCompleteWhen((_runOneStep OR _runAllSteps) AND _finishStep);

    IF _runOneStep THEN
        _runOneStep := FALSE;
        RETURN;
    END_IF
END_IF

IF SUPER^.Step(67, TRUE, 'Step number 67') THEN
    SUPER^.StepCompleteWhen((_runOneStep OR _runAllSteps) AND _finishStep);

    IF _runOneStep THEN
        _runOneStep := FALSE;
        RETURN;
    END_IF
END_IF

IF SUPER^.Step(68, TRUE, 'Step number 68') THEN
    SUPER^.StepCompleteWhen((_runOneStep OR _runAllSteps) AND _finishStep);

    IF _runOneStep THEN
        _runOneStep := FALSE;
        RETURN;
    END_IF
END_IF

IF SUPER^.Step(69, TRUE, 'Step number 69') THEN
    SUPER^.StepCompleteWhen((_runOneStep OR _runAllSteps) AND _finishStep);

    IF _runOneStep THEN
        _runOneStep := FALSE;
        RETURN;
    END_IF
END_IF

IF SUPER^.Step(70, TRUE, 'Step number 70') THEN
    SUPER^.StepCompleteWhen((_runOneStep OR _runAllSteps) AND _finishStep);

    IF _runOneStep THEN
        _runOneStep := FALSE;
        RETURN;
    END_IF
END_IF

IF SUPER^.Step(71, TRUE, 'Step number 71') THEN
    SUPER^.StepCompleteWhen((_runOneStep OR _runAllSteps) AND _finishStep);

    IF _runOneStep THEN
        _runOneStep := FALSE;
        RETURN;
    END_IF
END_IF

IF SUPER^.Step(72, TRUE, 'Step number 72') THEN
    SUPER^.StepCompleteWhen((_runOneStep OR _runAllSteps) AND _finishStep);

    IF _runOneStep THEN
        _runOneStep := FALSE;
        RETURN;
    END_IF
END_IF

IF SUPER^.Step(73, TRUE, 'Step number 73') THEN
    SUPER^.StepCompleteWhen((_runOneStep OR _runAllSteps) AND _finishStep);

    IF _runOneStep THEN
        _runOneStep := FALSE;
        RETURN;
    END_IF
END_IF

IF SUPER^.Step(74, TRUE, 'Step number 74') THEN
    SUPER^.StepCompleteWhen((_runOneStep OR _runAllSteps) AND _finishStep);

    IF _runOneStep THEN
        _runOneStep := FALSE;
        RETURN;
    END_IF
END_IF

IF SUPER^.Step(75, TRUE, 'Step number 75') THEN
    SUPER^.StepCompleteWhen((_runOneStep OR _runAllSteps) AND _finishStep);

    IF _runOneStep THEN
        _runOneStep := FALSE;
        RETURN;
    END_IF
END_IF

IF SUPER^.Step(76, TRUE, 'Step number 76') THEN
    SUPER^.StepCompleteWhen((_runOneStep OR _runAllSteps) AND _finishStep);

    IF _runOneStep THEN
        _runOneStep := FALSE;
        RETURN;
    END_IF
END_IF

IF SUPER^.Step(77, TRUE, 'Step number 77') THEN
    SUPER^.StepCompleteWhen((_runOneStep OR _runAllSteps) AND _finishStep);

    IF _runOneStep THEN
        _runOneStep := FALSE;
        RETURN;
    END_IF
END_IF

IF SUPER^.Step(78, TRUE, 'Step number 78') THEN
    SUPER^.StepCompleteWhen((_runOneStep OR _runAllSteps) AND _finishStep);

    IF _runOneStep THEN
        _runOneStep := FALSE;
        RETURN;
    END_IF
END_IF

IF SUPER^.Step(79, TRUE, 'Step number 79') THEN
    SUPER^.StepCompleteWhen((_runOneStep OR _runAllSteps) AND _finishStep);

    IF _runOneStep THEN
        _runOneStep := FALSE;
        RETURN;
    END_IF
END_IF

IF SUPER^.Step(80, TRUE, 'Step number 80') THEN
    SUPER^.StepCompleteWhen((_runOneStep OR _runAllSteps) AND _finishStep);

    IF _runOneStep THEN
        _runOneStep := FALSE;
        RETURN;
    END_IF
END_IF

IF SUPER^.Step(81, TRUE, 'Step number 81') THEN
    SUPER^.StepCompleteWhen((_runOneStep OR _runAllSteps) AND _finishStep);

    IF _runOneStep THEN
        _runOneStep := FALSE;
        RETURN;
    END_IF
END_IF

